# B&R Automation Studio project BenchEDM_AS6 (part 7)

#### Seq_INIT_X.st - not listed in the package file held
```iecst
ACTION Seq_INIT_X:

	TC_Seq_Add(ADR(JSONStrings),ADR('{"driver":"AB","inst":"VX_0","type":"C","ident":"ERRORRESET","enable":"TRUE"}'));
	TC_Seq_Add(ADR(JSONStrings),ADR('{"driver":"AB","inst":"VX_0","type":"W","ident":"NOERROR","time":"10.0"}'));
	TC_Seq_Add(ADR(JSONStrings),ADR('{"driver":"AB","inst":"VX_0","type":"C","ident":"ERRORRESET","enable":"FALSE"}'));
	TC_Seq_Add(ADR(JSONStrings),ADR('{"driver":"AB","inst":"VX_0","type":"M","ident":"ERROR","enable":"TRUE","sev":"4","time":"0.0"}'));
	TC_Seq_Add(ADR(JSONStrings),ADR('{"driver":"AB","inst":"VX_0","type":"W","ident":"READYTOPOWERON","time":"10.0"}'));
	TC_Seq_Add(ADR(JSONStrings),ADR('{"driver":"AB","inst":"VX_0","type":"C","ident":"POWER","enable":"TRUE"}'));
	TC_Seq_Add(ADR(JSONStrings),ADR('{"driver":"AB","inst":"VX_0","type":"W","ident":"POWERON","time":"5.0"}'));
	TC_Seq_Add(ADR(JSONStrings),ADR('{"driver":"AB","inst":"VX_0","type":"M","ident":"NOTPOWERON","enable":"TRUE","sev":"4","time":"0.0"}'));
	TC_Seq_Add(ADR(JSONStrings),ADR('{"driver":"AB","inst":"VX_0","type":"C","ident":"HOME","enable":"TRUE"}'));
	TC_Seq_Add(ADR(JSONStrings),ADR('{"driver":"AB","inst":"VX_0","type":"W","ident":"ISHOMED","time":"5.0"}'));
	TC_Seq_Add(ADR(JSONStrings),ADR('{"driver":"AB","inst":"VX_0","type":"C","ident":"HOME","enable":"FALSE"}'));

	TC_Seq_Add(ADR(JSONStrings),ADR('{"driver":"AB","inst":"RX0_0","type":"C","ident":"ERRORRESET","enable":"TRUE"}'));
	TC_Seq_Add(ADR(JSONStrings),ADR('{"driver":"AB","inst":"RX0_0","type":"W","ident":"NOERROR","time":"10.0"}'));
	TC_Seq_Add(ADR(JSONStrings),ADR('{"driver":"AB","inst":"RX0_0","type":"C","ident":"ERRORRESET","enable":"FALSE"}'));
	TC_Seq_Add(ADR(JSONStrings),ADR('{"driver":"AB","inst":"RX0_0","type":"M","ident":"ERROR","enable":"TRUE","sev":"4","time":"0.0"}'));
	TC_Seq_Add(ADR(JSONStrings),ADR('{"driver":"AB","inst":"RX0_0","type":"W","ident":"READYTOPOWERON","time":"10.0"}'));
	TC_Seq_Add(ADR(JSONStrings),ADR('{"driver":"AB","inst":"RX0_0","type":"C","ident":"POWER","enable":"TRUE"}'));
	TC_Seq_Add(ADR(JSONStrings),ADR('{"driver":"AB","inst":"RX0_0","type":"W","ident":"POWERON","time":"5.0"}'));
	TC_Seq_Add(ADR(JSONStrings),ADR('{"driver":"AB","inst":"RX0_0","type":"M","ident":"NOTPOWERON","enable":"TRUE","sev":"4","time":"0.0"}'));
	TC_Seq_Add(ADR(JSONStrings),ADR('{"driver":"AB","inst":"RX0_0","type":"C","ident":"HOME","enable":"TRUE"}'));
	TC_Seq_Add(ADR(JSONStrings),ADR('{"driver":"AB","inst":"RX0_0","type":"W","ident":"ISHOMED","time":"5.0"}'));
	TC_Seq_Add(ADR(JSONStrings),ADR('{"driver":"AB","inst":"RX0_0","type":"C","ident":"HOME","enable":"FALSE"}'));

	TC_Seq_Add(ADR(JSONStrings),ADR('{"driver":"CS","inst":"RX0_0","type":"C","ident":"ERRORRESET","enable":"TRUE"}'));
	TC_Seq_Add(ADR(JSONStrings),ADR('{"driver":"CS","inst":"RX0_0","type":"W","ident":"NOERROR","time":"10.0"}'));
	TC_Seq_Add(ADR(JSONStrings),ADR('{"driver":"CS","inst":"RX0_0","type":"C","ident":"ERRORRESET","enable":"FALSE"}'));
	TC_Seq_Add(ADR(JSONStrings),ADR('{"driver":"CS","inst":"RX0_0","type":"M","ident":"ERROR","enable":"TRUE","sev":"4","time":"0.0"}'));
	TC_Seq_Add(ADR(JSONStrings),ADR('{"driver":"CS","inst":"RX0_0","type":"W","ident":"AXISREADY","time":"10.0"}'));
	TC_Seq_Add(ADR(JSONStrings),ADR('{"driver":"CS","inst":"RX0_0","type":"C","ident":"MOVECYCLICPOSITION","enable":"TRUE","par":{"CyclicPositionSource":"<SD>0"}}'));
	TC_Seq_Add(ADR(JSONStrings),ADR('{"driver":"CS","inst":"RX0_0","type":"W","ident":"MOVECYCLICPOSITIONACTIVE","time":"10.0"}'));
	TC_Seq_Add(ADR(JSONStrings),ADR('{"driver":"CS","inst":"RX0_0","type":"M","ident":"NOTMOVECYCLICPOSITIONACTIVE","enable":"TRUE","sev":"4","time":"0.0"}'));

END_ACTION
```

#### Seq_INIT_Y.st - not listed in the package file held
```iecst
ACTION Seq_INIT_Y:

	TC_Seq_Add(ADR(JSONStrings),ADR('{"driver":"AB","inst":"VY_0","type":"C","ident":"ERRORRESET","enable":"TRUE"}'));
	TC_Seq_Add(ADR(JSONStrings),ADR('{"driver":"AB","inst":"VY_0","type":"W","ident":"NOERROR","time":"10.0"}'));
	TC_Seq_Add(ADR(JSONStrings),ADR('{"driver":"AB","inst":"VY_0","type":"C","ident":"ERRORRESET","enable":"FALSE"}'));
	TC_Seq_Add(ADR(JSONStrings),ADR('{"driver":"AB","inst":"VY_0","type":"M","ident":"ERROR","enable":"TRUE","sev":"4","time":"0.0"}'));
	TC_Seq_Add(ADR(JSONStrings),ADR('{"driver":"AB","inst":"VY_0","type":"W","ident":"READYTOPOWERON","time":"10.0"}'));
	TC_Seq_Add(ADR(JSONStrings),ADR('{"driver":"AB","inst":"VY_0","type":"C","ident":"POWER","enable":"TRUE"}'));
	TC_Seq_Add(ADR(JSONStrings),ADR('{"driver":"AB","inst":"VY_0","type":"W","ident":"POWERON","time":"5.0"}'));
	TC_Seq_Add(ADR(JSONStrings),ADR('{"driver":"AB","inst":"VY_0","type":"M","ident":"NOTPOWERON","enable":"TRUE","sev":"4","time":"0.0"}'));
	TC_Seq_Add(ADR(JSONStrings),ADR('{"driver":"AB","inst":"VY_0","type":"C","ident":"HOME","enable":"TRUE"}'));
	TC_Seq_Add(ADR(JSONStrings),ADR('{"driver":"AB","inst":"VY_0","type":"W","ident":"ISHOMED","time":"5.0"}'));
	TC_Seq_Add(ADR(JSONStrings),ADR('{"driver":"AB","inst":"VY_0","type":"C","ident":"HOME","enable":"FALSE"}'));

	TC_Seq_Add(ADR(JSONStrings),ADR('{"driver":"AB","inst":"RY0_0","type":"C","ident":"ERRORRESET","enable":"TRUE"}'));
	TC_Seq_Add(ADR(JSONStrings),ADR('{"driver":"AB","inst":"RY0_0","type":"W","ident":"NOERROR","time":"10.0"}'));
	TC_Seq_Add(ADR(JSONStrings),ADR('{"driver":"AB","inst":"RY0_0","type":"C","ident":"ERRORRESET","enable":"FALSE"}'));
	TC_Seq_Add(ADR(JSONStrings),ADR('{"driver":"AB","inst":"RY0_0","type":"M","ident":"ERROR","enable":"TRUE","sev":"4","time":"0.0"}'));
	TC_Seq_Add(ADR(JSONStrings),ADR('{"driver":"AB","inst":"RY0_0","type":"W","ident":"READYTOPOWERON","time":"10.0"}'));
	TC_Seq_Add(ADR(JSONStrings),ADR('{"driver":"AB","inst":"RY0_0","type":"C","ident":"POWER","enable":"TRUE"}'));
	TC_Seq_Add(ADR(JSONStrings),ADR('{"driver":"AB","inst":"RY0_0","type":"W","ident":"POWERON","time":"5.0"}'));
	TC_Seq_Add(ADR(JSONStrings),ADR('{"driver":"AB","inst":"RY0_0","type":"M","ident":"NOTPOWERON","enable":"TRUE","sev":"4","time":"0.0"}'));
	TC_Seq_Add(ADR(JSONStrings),ADR('{"driver":"AB","inst":"RY0_0","type":"C","ident":"HOME","enable":"TRUE"}'));
	TC_Seq_Add(ADR(JSONStrings),ADR('{"driver":"AB","inst":"RY0_0","type":"W","ident":"ISHOMED","time":"5.0"}'));
	TC_Seq_Add(ADR(JSONStrings),ADR('{"driver":"AB","inst":"RY0_0","type":"C","ident":"HOME","enable":"FALSE"}'));

	TC_Seq_Add(ADR(JSONStrings),ADR('{"driver":"CS","inst":"RY0_0","type":"C","ident":"ERRORRESET","enable":"TRUE"}'));
	TC_Seq_Add(ADR(JSONStrings),ADR('{"driver":"CS","inst":"RY0_0","type":"W","ident":"NOERROR","time":"10.0"}'));
	TC_Seq_Add(ADR(JSONStrings),ADR('{"driver":"CS","inst":"RY0_0","type":"C","ident":"ERRORRESET","enable":"FALSE"}'));
	TC_Seq_Add(ADR(JSONStrings),ADR('{"driver":"CS","inst":"RY0_0","type":"M","ident":"ERROR","enable":"TRUE","sev":"4","time":"0.0"}'));
	TC_Seq_Add(ADR(JSONStrings),ADR('{"driver":"CS","inst":"RY0_0","type":"W","ident":"AXISREADY","time":"10.0"}'));
	TC_Seq_Add(ADR(JSONStrings),ADR('{"driver":"CS","inst":"RY0_0","type":"C","ident":"MOVECYCLICPOSITION","enable":"TRUE","par":{"CyclicPositionSource":"<SD>0"}}'));
	TC_Seq_Add(ADR(JSONStrings),ADR('{"driver":"CS","inst":"RY0_0","type":"W","ident":"MOVECYCLICPOSITIONACTIVE","time":"10.0"}'));
	TC_Seq_Add(ADR(JSONStrings),ADR('{"driver":"CS","inst":"RY0_0","type":"M","ident":"NOTMOVECYCLICPOSITIONACTIVE","enable":"TRUE","sev":"4","time":"0.0"}'));

END_ACTION
```

#### Seq_INIT_Z.st - not listed in the package file held
```iecst
ACTION Seq_INIT_Z:

	TC_Seq_Add(ADR(JSONStrings),ADR('{"driver":"AB","inst":"VZ_0","type":"C","ident":"ERRORRESET","enable":"TRUE"}'));
	TC_Seq_Add(ADR(JSONStrings),ADR('{"driver":"AB","inst":"VZ_0","type":"W","ident":"NOERROR","time":"10.0"}'));
	TC_Seq_Add(ADR(JSONStrings),ADR('{"driver":"AB","inst":"VZ_0","type":"C","ident":"ERRORRESET","enable":"FALSE"}'));
	TC_Seq_Add(ADR(JSONStrings),ADR('{"driver":"AB","inst":"VZ_0","type":"M","ident":"ERROR","enable":"TRUE","sev":"4","time":"0.0"}'));
	TC_Seq_Add(ADR(JSONStrings),ADR('{"driver":"AB","inst":"VZ_0","type":"W","ident":"READYTOPOWERON","time":"10.0"}'));
	TC_Seq_Add(ADR(JSONStrings),ADR('{"driver":"AB","inst":"VZ_0","type":"C","ident":"POWER","enable":"TRUE"}'));
	TC_Seq_Add(ADR(JSONStrings),ADR('{"driver":"AB","inst":"VZ_0","type":"W","ident":"POWERON","time":"5.0"}'));
	TC_Seq_Add(ADR(JSONStrings),ADR('{"driver":"AB","inst":"VZ_0","type":"M","ident":"NOTPOWERON","enable":"TRUE","sev":"4","time":"0.0"}'));
	TC_Seq_Add(ADR(JSONStrings),ADR('{"driver":"AB","inst":"VZ_0","type":"C","ident":"HOME","enable":"TRUE"}'));
	TC_Seq_Add(ADR(JSONStrings),ADR('{"driver":"AB","inst":"VZ_0","type":"W","ident":"ISHOMED","time":"5.0"}'));
	TC_Seq_Add(ADR(JSONStrings),ADR('{"driver":"AB","inst":"VZ_0","type":"C","ident":"HOME","enable":"FALSE"}'));

	TC_Seq_Add(ADR(JSONStrings),ADR('{"driver":"AB","inst":"RZ0_0","type":"C","ident":"ERRORRESET","enable":"TRUE"}'));
	TC_Seq_Add(ADR(JSONStrings),ADR('{"driver":"AB","inst":"RZ0_0","type":"W","ident":"NOERROR","time":"10.0"}'));
	TC_Seq_Add(ADR(JSONStrings),ADR('{"driver":"AB","inst":"RZ0_0","type":"C","ident":"ERRORRESET","enable":"FALSE"}'));
	TC_Seq_Add(ADR(JSONStrings),ADR('{"driver":"AB","inst":"RZ0_0","type":"M","ident":"ERROR","enable":"TRUE","sev":"4","time":"0.0"}'));
	TC_Seq_Add(ADR(JSONStrings),ADR('{"driver":"AB","inst":"RZ0_0","type":"W","ident":"READYTOPOWERON","time":"10.0"}'));
	TC_Seq_Add(ADR(JSONStrings),ADR('{"driver":"AB","inst":"RZ0_0","type":"C","ident":"POWER","enable":"TRUE"}'));
	TC_Seq_Add(ADR(JSONStrings),ADR('{"driver":"AB","inst":"RZ0_0","type":"W","ident":"POWERON","time":"5.0"}'));
	TC_Seq_Add(ADR(JSONStrings),ADR('{"driver":"AB","inst":"RZ0_0","type":"M","ident":"NOTPOWERON","enable":"TRUE","sev":"4","time":"0.0"}'));
	TC_Seq_Add(ADR(JSONStrings),ADR('{"driver":"AB","inst":"RZ0_0","type":"C","ident":"HOME","enable":"TRUE"}'));
	TC_Seq_Add(ADR(JSONStrings),ADR('{"driver":"AB","inst":"RZ0_0","type":"W","ident":"ISHOMED","time":"5.0"}'));
	TC_Seq_Add(ADR(JSONStrings),ADR('{"driver":"AB","inst":"RZ0_0","type":"C","ident":"HOME","enable":"FALSE"}'));

	TC_Seq_Add(ADR(JSONStrings),ADR('{"driver":"CS","inst":"RZ0_0","type":"C","ident":"ERRORRESET","enable":"TRUE"}'));
	TC_Seq_Add(ADR(JSONStrings),ADR('{"driver":"CS","inst":"RZ0_0","type":"W","ident":"NOERROR","time":"10.0"}'));
	TC_Seq_Add(ADR(JSONStrings),ADR('{"driver":"CS","inst":"RZ0_0","type":"C","ident":"ERRORRESET","enable":"FALSE"}'));
	TC_Seq_Add(ADR(JSONStrings),ADR('{"driver":"CS","inst":"RZ0_0","type":"M","ident":"ERROR","enable":"TRUE","sev":"4","time":"0.0"}'));
	TC_Seq_Add(ADR(JSONStrings),ADR('{"driver":"CS","inst":"RZ0_0","type":"W","ident":"AXISREADY","time":"10.0"}'));
	TC_Seq_Add(ADR(JSONStrings),ADR('{"driver":"CS","inst":"RZ0_0","type":"C","ident":"MOVECYCLICPOSITION","enable":"TRUE","par":{"CyclicPositionSource":"<SD>0"}}'));
	TC_Seq_Add(ADR(JSONStrings),ADR('{"driver":"CS","inst":"RZ0_0","type":"W","ident":"MOVECYCLICPOSITIONACTIVE","time":"10.0"}'));
	TC_Seq_Add(ADR(JSONStrings),ADR('{"driver":"CS","inst":"RZ0_0","type":"M","ident":"NOTMOVECYCLICPOSITIONACTIVE","enable":"TRUE","sev":"4","time":"0.0"}'));

END_ACTION
```

### Program Logical/Process/OutputMan (IEC)

#### Main.st - Init, cyclic, exit code
```iecst
PROGRAM _INIT

END_PROGRAM

PROGRAM _CYCLIC

	OMD_CN;
	OMD_AB;
	OMD_CS;
	OMD_MR;
	OMD_BX;
	gDriver.ResetAll := FALSE;

//BX18

	IF (gIO.BX18.TC_IO_DO_Enable.Forcing.On AND gIO.BX18.TC_IO_DO_Enable.Forcing.Off) OR NOT gIO.ForceEnable THEN
		gIO.BX18.TC_IO_DO_Enable.Forcing.On									:= FALSE;
		gIO.BX18.TC_IO_DO_Enable.Forcing.Off								:= FALSE;
	END_IF;
	gIO.BX18.TC_IO_DO_Enable(Par := gPar.IO.BX18.TC_IO_DO_Enable);

	IF (gIO.BX18.TC_IO_DO_ISOFreqMode.Forcing.On AND gIO.BX18.TC_IO_DO_ISOFreqMode.Forcing.Off) OR NOT gIO.ForceEnable THEN
		gIO.BX18.TC_IO_DO_ISOFreqMode.Forcing.On							:= FALSE;
		gIO.BX18.TC_IO_DO_ISOFreqMode.Forcing.Off							:= FALSE;
	END_IF;
	gIO.BX18.TC_IO_DO_ISOFreqMode(Par := gPar.IO.BX18.TC_IO_DO_ISOFreqMode);

	IF (gIO.BX18.TC_IO_DO_EdgeFindMode.Forcing.On AND gIO.BX18.TC_IO_DO_EdgeFindMode.Forcing.Off) OR NOT gIO.ForceEnable THEN
		gIO.BX18.TC_IO_DO_EdgeFindMode.Forcing.On							:= FALSE;
		gIO.BX18.TC_IO_DO_EdgeFindMode.Forcing.Off							:= FALSE;
	END_IF;
	gIO.BX18.TC_IO_DO_EdgeFindMode(Par := gPar.IO.BX18.TC_IO_DO_EdgeFindMode);

	IF (gIO.BX18.TC_IO_DO_ElectrodePositiveMode.Forcing.On AND gIO.BX18.TC_IO_DO_ElectrodePositiveMode.Forcing.Off) OR NOT gIO.ForceEnable THEN
		gIO.BX18.TC_IO_DO_ElectrodePositiveMode.Forcing.On					:= FALSE;
		gIO.BX18.TC_IO_DO_ElectrodePositiveMode.Forcing.Off					:= FALSE;
	END_IF;
	gIO.BX18.TC_IO_DO_ElectrodePositiveMode(Par := gPar.IO.BX18.TC_IO_DO_ElectrodePositiveMode);

	IF (gIO.BX18.TC_IO_DO_ChangeRequest.Forcing.On AND gIO.BX18.TC_IO_DO_ChangeRequest.Forcing.Off) OR NOT gIO.ForceEnable THEN
		gIO.BX18.TC_IO_DO_ChangeRequest.Forcing.On							:= FALSE;
		gIO.BX18.TC_IO_DO_ChangeRequest.Forcing.Off							:= FALSE;
	END_IF;
	gIO.BX18.TC_IO_DO_ChangeRequest(Par := gPar.IO.BX18.TC_IO_DO_ChangeRequest);

	IF (gIO.BX18.TC_IO_AO_OnTime.Forcing.On AND gIO.BX18.TC_IO_AO_OnTime.Forcing.Off) OR NOT gIO.ForceEnable THEN
		gIO.BX18.TC_IO_AO_OnTime.Forcing.On									:= FALSE;
		gIO.BX18.TC_IO_AO_OnTime.Forcing.Off								:= FALSE;
	END_IF;
	gIO.BX18.TC_IO_AO_OnTime(Par := gPar.IO.BX18.TC_IO_AO_OnTime, VarType := TC_IO_ANALOG_TYPE_UINT);

	IF (gIO.BX18.TC_IO_AO_OffTime.Forcing.On AND gIO.BX18.TC_IO_AO_OffTime.Forcing.Off) OR NOT gIO.ForceEnable THEN
		gIO.BX18.TC_IO_AO_OffTime.Forcing.On								:= FALSE;
		gIO.BX18.TC_IO_AO_OffTime.Forcing.Off								:= FALSE;
	END_IF;
	gIO.BX18.TC_IO_AO_OffTime(Par := gPar.IO.BX18.TC_IO_AO_OffTime, VarType := TC_IO_ANALOG_TYPE_UINT);

	IF (gIO.BX18.TC_IO_AO_Current.Forcing.On AND gIO.BX18.TC_IO_AO_Current.Forcing.Off) OR NOT gIO.ForceEnable THEN
		gIO.BX18.TC_IO_AO_Current.Forcing.On								:= FALSE;
		gIO.BX18.TC_IO_AO_Current.Forcing.Off								:= FALSE;
	END_IF;
	gIO.BX18.TC_IO_AO_Current(Par := gPar.IO.BX18.TC_IO_AO_Current, VarType := TC_IO_ANALOG_TYPE_UINT);

	gIO.BX18.Outputs_control.0												:= gIO.BX18.TC_IO_DO_Enable.Signal.IOMapping;
	gIO.BX18.Outputs_control.1												:= gIO.BX18.TC_IO_DO_ISOFreqMode.Signal.IOMapping;
	gIO.BX18.Outputs_control.2												:= gIO.BX18.TC_IO_DO_EdgeFindMode.Signal.IOMapping;
	gIO.BX18.Outputs_control.3												:= gIO.BX18.TC_IO_DO_ElectrodePositiveMode.Signal.IOMapping;
	gIO.BX18.Outputs_control.4												:= gIO.BX18.TC_IO_DO_ChangeRequest.Signal.IOMapping;
	gIO.BX18.Outputs_onTime													:= gIO.BX18.TC_IO_AO_OnTime.Signal.IOMapping.VarUINT;
	gIO.BX18.Outputs_offTime												:= gIO.BX18.TC_IO_AO_OffTime.Signal.IOMapping.VarUINT;
	gIO.BX18.Outputs_current												:= gIO.BX18.TC_IO_AO_Current.Signal.IOMapping.VarUINT;
//Motion
	gIO.Motion.SetPosition 													:= LREAL_TO_DINT(gDriver.AB[DRIVER_INST_AB_RZ_0_0].Status.Position*200.0); //200.0 is the scaling to get 1mm travel for 1000 dip switch setting on stepper drive
	gIO.Motion.StepDelay 													:= STEPDELAY;
	gIO.Motion.ENABLE														:= gIO.Motion.ModuleOK;
	gIO.Motion.SwitchedOn													:= gIO.Motion.ENABLED AND gIO.Motion.SwitchOn AND gIO.Safety.TC_IO_DI_ESTOP.Signal.Filtered;
	gIO.Motion.Home															:= EDGEPOS(gDriver.AB[DRIVER_INST_AB_RZ_0_0].MpAxisBasic_0.IsHomed);
//MbRTU VFDs
	FOR i := 0 TO MAX_VFD_IDX DO
		gIO.VFD[i].DataWrite[0] := gIO.VFD[i].CMD;
		gIO.VFD[i].DataWrite[1] := gIO.VFD[i].LFRD;
		FOR j := 0 TO MAX_VFD_DATA_READ_IDX DO
			gIO.VFD[i].EventRead[j]											:= TRUE;
		END_FOR;
		gIO.VFD[i].CTON_AutoWrite(IN := NOT gIO.VFD[i].CTON_AutoWrite.Q, PT := T#500ms);
		FOR j := 0 TO MAX_VFD_DATA_WRITE_IDX DO
			IF gIO.VFD[i].DataWriteCmp[j] <> gIO.VFD[i].DataWrite[j] OR gIO.VFD[i].CTON_AutoWrite.Q THEN
				gIO.VFD[i].EventWrite[j]									:= TRUE;
				gIO.VFD[i].DataWriteCmp[j] 									:= gIO.VFD[i].DataWrite[j];
			END_IF;
		END_FOR;
		gIO.VFD[i].ETA := gIO.VFD[i].DataRead[0];
		gIO.VFD[i].RFRD := gIO.VFD[i].DataRead[1];
		gIO.VFD[i].LFT := gIO.VFD[i].DataRead[2];
	END_FOR;

END_PROGRAM

PROGRAM _EXIT

END_PROGRAM
```

#### OMD_IN.st
```iecst
ACTION OMD_IN:

//	FOR i := 0 TO MAX_DRIVER_IN_IDX DO
//		IF NOT gDriver.IN[i].FirstScanComplete THEN
//			gDriver.IN[i].FirstScanComplete 													:= TRUE;
//
//			gDriver.IN[i].DefaultPar.DI_Estop_Par.FilterOnTime									:= 50.0;							//LR
//			gDriver.IN[i].DefaultPar.DI_Estop_Par.FilterOffTime									:= 50.0;							//LR
//			gDriver.IN[i].DefaultPar.DI_Estop_Par.InvertedIOMapping								:= FALSE;							//BO
//			gDriver.IN[i].DefaultPar.DI_Estop_Forcing.On										:= FALSE;							//BO
//			gDriver.IN[i].DefaultPar.DI_Estop_Forcing.Off										:= FALSE;							//BO
//			gDriver.IN[i].DefaultPar.DI_Estop_Sim.Active										:= gSim.Full OR gSim.IO;			//BO
//			gDriver.IN[i].DefaultPar.DI_Estop_Sim.Logical										:= FALSE;							//BO
//
//			brsmemcpy(ADR(gDriver.IN[i].Par),ADR(gDriver.IN[i].DefaultPar),SIZEOF(gDriver.IN[i].Par));
//		END_IF;
//
//		brsmemset(ADR(gDriver.IN[i].Sev),0,SIZEOF(gDriver.IN[i].Sev));
//		brsmemset(ADR(gDriver.IN[i].Status),0,SIZEOF(gDriver.IN[i].Status));
//		FOR j := 0 TO MAX_DRIVER_IN_MON_IDX DO
//			IF gDriver.IN[i].Par.Mon[j].Enable THEN
//				IF gDriver.IN[i].Mon[j] THEN
//					gDriver.IN[i].CTON_Mon[j](IN := TRUE, PT := LREAL_TO_TIME(gDriver.IN[i].Par.Mon[j].Time*1000.0));
//					IF gDriver.IN[i].CTON_Mon[j].Q THEN
//						gDriver.IN[i].Sev[j] := gDriver.IN[i].Par.Mon[j].Sev;
//						IF gDriver.IN[i].Status.Severity < gDriver.IN[i].Sev[j] THEN
//							gDriver.IN[i].Status.Severity := gDriver.IN[i].Sev[j];
//						END_IF;
//					END_IF;
//				ELSE
//					gDriver.IN[i].CTON_Mon[j](IN := FALSE);
//					gDriver.IN[i].Sev[j] := 0;
//				END_IF;
//			ELSE
//				gDriver.IN[i].CTON_Mon[j](IN := FALSE);
//				gDriver.IN[i].Sev[j] := 0;
//			END_IF;
//		END_FOR;
//		IF gDriver.IN[i].Cmd[C_IN_RESET] THEN
//			gDriver.IN[i].Cmd[C_IN_RESET] := FALSE;
//			brsmemset(ADR(gDriver.IN[i].Cmd),0,SIZEOF(gDriver.IN[i].Cmd));
//			brsmemset(ADR(gDriver.IN[i].Sev),0,SIZEOF(gDriver.IN[i].Sev));
//			brsmemset(ADR(gDriver.IN[i].Status),0,SIZEOF(gDriver.IN[i].Status));
//			brsmemcpy(ADR(gDriver.IN[i].Par),ADR(gDriver.IN[i].DefaultPar),SIZEOF(gDriver.IN[i].Par));
//		END_IF;
//		IF gDriver.IN[i].Cmd[C_IN_CLEARCMD] THEN
//			gDriver.IN[i].Cmd[C_IN_CLEARCMD] := FALSE;
//			brsmemset(ADR(gDriver.IN[i].Cmd),0,SIZEOF(gDriver.IN[i].Cmd));
//		END_IF;
//		IF gDriver.IN[i].Cmd[C_IN_CLEARMON] THEN
//			gDriver.IN[i].Cmd[C_IN_CLEARMON] := FALSE;
//			brsmemset(ADR(gDriver.IN[i].Status.Severity),0,SIZEOF(gDriver.IN[i].Status.Severity));
//			brsmemset(ADR(gDriver.IN[i].Sev),0,SIZEOF(gDriver.IN[i].Sev));
//			brsmemset(ADR(gDriver.IN[i].Par.Mon),0,SIZEOF(gDriver.IN[i].Par.Mon));
//		END_IF;
//		IF gDriver.IN[i].Cmd[C_IN_DEFAULTMON] THEN
//			gDriver.IN[i].Cmd[C_IN_DEFAULTMON] := FALSE;
//			brsmemcpy(ADR(gDriver.IN[i].Par.Mon),ADR(gDriver.IN[i].DefaultPar.Mon),SIZEOF(gDriver.IN[i].Par.Mon));
//		END_IF;
//		IF gDriver.IN[i].Cmd[C_IN_CLEARPAR] THEN
//			gDriver.IN[i].Cmd[C_IN_CLEARPAR] := FALSE;
//			brsmemset(ADR(gDriver.IN[i].Par),0,SIZEOF(gDriver.IN[i].Par));
//		END_IF;
//		IF gDriver.IN[i].Cmd[C_IN_DEFAULTPAR] THEN
//			gDriver.IN[i].Cmd[C_IN_DEFAULTPAR] := FALSE;
//			brsmemcpy(ADR(gDriver.IN[i].Par),ADR(gDriver.IN[i].DefaultPar),SIZEOF(gDriver.IN[i].Par));
//		END_IF;
//		IF gDriver.IN[i].Cmd[C_IN_FORCEENABLE] THEN
//			gDriver.IN[i].Cmd[C_IN_FORCEENABLE] := FALSE;
//			gDriver.IN[i].Par.ForceEnable := TRUE;
//		END_IF;
//		IF gDriver.IN[i].Cmd[C_IN_FORCEDISABLE] THEN
//			gDriver.IN[i].Cmd[C_IN_FORCEDISABLE] := FALSE;
//			gDriver.IN[i].Par.ForceEnable := FALSE;
//		END_IF;
//
//		IF NOT gDriver.IN[i].Par.ForceEnable OR (gDriver.IN[i].Par.DI_Estop_Forcing.On AND gDriver.IN[i].Par.DI_Estop_Forcing.Off) THEN
//			gDriver.IN[i].Par.DI_Estop_Forcing.On := FALSE;
//			gDriver.IN[i].Par.DI_Estop_Forcing.Off := FALSE;
//		END_IF;
//		gDriver.IN[i].DI_Estop(Forcing := gDriver.IN[i].Par.DI_Estop_Forcing, Par := gDriver.IN[i].Par.DI_Estop_Par, Sim := gDriver.IN[i].Par.DI_Estop_Sim);
//
//		gDriver.IN[i].Wait[W_IN_DI_ESTOP]				:= BOOL_TO_DINT(NOT gDriver.IN[i].DI_Estop.Signal.Filtered);
//
//		gDriver.IN[i].Mon[M_IN_ERROR]					:= gDriver.IN[i].MpAxisBasic_0.Error;
//	END_FOR;
//
////	McSwitchEnum :
////	(
////		mcSWITCH_OFF := 0,		 						(*State/Behavior selection switched off*)
////		mcSWITCH_ON := 1			 					(*State/Behavior selection switched on*)
////	);

END_ACTION
```

#### OMD_CN.st
```iecst
ACTION OMD_CN:

	gDriver.CN[DRIVER_INST_CN_0].MpLinkADR 																:= ADR(gCNC);
	gDriver.CN[DRIVER_INST_CN_0].OverrideSetpoint[0]													:= 100.0;
	gDriver.CN[DRIVER_INST_CN_0].OverrideSetpoint[1]													:= gDriver.BX[DRIVER_INST_BX_0].Status.OverrideFactor;
	gDriver.CN[DRIVER_INST_CN_0].RapidOverrideSetpoint[0]												:= 100.0;
	gDriver.CN[DRIVER_INST_CN_0].FeedrateOverrideSetpoint[0]											:= 100.0;

	FOR i := 0 TO MAX_DRIVER_CN_IDX DO
		IF NOT gDriver.CN[i].FirstScanComplete THEN
			gDriver.CN[i].FirstScanComplete 															:= TRUE;

			gDriver.CN[i].DefaultPar.CN.Block															:= '';								//ST
			gDriver.CN[i].DefaultPar.CN.Jog.CoordSystem													:= 0;								//UD
			gDriver.CN[i].DefaultPar.CN.Jog.PathLimits.Acceleration										:= 50.0;							//RR
			gDriver.CN[i].DefaultPar.CN.Jog.PathLimits.Deceleration										:= 50.0;							//RR
			gDriver.CN[i].DefaultPar.CN.Jog.PathLimits.Jerk												:= 0.0;								//RR
			gDriver.CN[i].DefaultPar.CN.Jog.PathLimits.Velocity											:= 10.0;							//RR
			gDriver.CN[i].DefaultPar.CN.MoveProgramOptions.InitProgram									:= '';								//ST
			gDriver.CN[i].DefaultPar.CN.MoveProgramOptions.RepositioningParameter.AxisVelocityFactor	:= 10.0;							//RR
			gDriver.CN[i].DefaultPar.CN.MoveProgramOptions.RepositioningParameter.String				:= '';								//ST
			gDriver.CN[i].DefaultPar.CN.MoveProgramOptions.RepositioningParameter.Type					:= mcPRGRP_SINGLE_AXIS;				//McPrgAxesReposTypeEnum
			gDriver.CN[i].DefaultPar.CN.MoveProgramOptions.SaveRestartData								:= mcSWITCH_OFF;					//McSwitchEnum
			gDriver.CN[i].DefaultPar.CN.MoveProgramOptions.StartMode									:= mcPRGSM_NON_MODAL;				//McPrgStartModeEnum
			gDriver.CN[i].DefaultPar.CN.MoveProgramOptions.StartPointParameter							:= 0.0;								//LR
			gDriver.CN[i].DefaultPar.CN.MoveProgramOptions.StartPointType								:= mcPRGSP_STANDARD;				//McPrgStartPointEnum
			gDriver.CN[i].DefaultPar.CN.ProgramName														:= '';								//ST
			gDriver.CN[i].DefaultPar.FeedrateOverrideSource												:= 0;								//SD
			gDriver.CN[i].DefaultPar.OverrideSource														:= 0;								//SD
			gDriver.CN[i].DefaultPar.RapidOverrideSource												:= 0;								//SD
			brsmemcpy(ADR(gDriver.CN[i].Par),ADR(gDriver.CN[i].DefaultPar),SIZEOF(gDriver.CN[i].Par));
		ELSIF NOT gDriver.CN[i].ParametersLoaded AND gMain.Services.Recipes.Out.ParametersReady THEN
			gDriver.CN[i].ParametersLoaded := TRUE;
			brsmemcpy(ADR(gDriver.CN[i].Par),ADR(gPar.Driver.CN[i]),SIZEOF(gDriver.CN[i].Par));
		END_IF;

		brsmemset(ADR(gDriver.CN[i].Sev),0,SIZEOF(gDriver.CN[i].Sev));
		brsmemset(ADR(gDriver.CN[i].Status),0,SIZEOF(gDriver.CN[i].Status));
		FOR j := 0 TO MAX_DRIVER_CN_MON_IDX DO
			IF gDriver.CN[i].Par.Mon[j].Enable THEN
				IF gDriver.CN[i].Mon[j] THEN
					gDriver.CN[i].CTON_Mon[j](IN := TRUE, PT := LREAL_TO_TIME(gDriver.CN[i].Par.Mon[j].Time*1000.0));
					IF gDriver.CN[i].CTON_Mon[j].Q THEN
						gDriver.CN[i].Sev[j] := gDriver.CN[i].Par.Mon[j].Sev;
						IF gDriver.CN[i].Status.Severity < gDriver.CN[i].Sev[j] THEN
							gDriver.CN[i].Status.Severity := gDriver.CN[i].Sev[j];
						END_IF;
					END_IF;
				ELSE
					gDriver.CN[i].CTON_Mon[j](IN := FALSE);
					gDriver.CN[i].Sev[j] := 0;
				END_IF;
			ELSE
				gDriver.CN[i].CTON_Mon[j](IN := FALSE);
				gDriver.CN[i].Sev[j] := 0;
			END_IF;
		END_FOR;
		IF gDriver.CN[i].Cmd[C_CN_RESET] OR gDriver.ResetAll THEN
			gDriver.CN[i].Cmd[C_CN_RESET] := FALSE;
			brsmemset(ADR(gDriver.CN[i].Mon),0,SIZEOF(gDriver.CN[i].Mon));
			brsmemset(ADR(gDriver.CN[i].Cmd),0,SIZEOF(gDriver.CN[i].Cmd));
			brsmemset(ADR(gDriver.CN[i].Sev),0,SIZEOF(gDriver.CN[i].Sev));
			brsmemset(ADR(gDriver.CN[i].Status),0,SIZEOF(gDriver.CN[i].Status));
		END_IF;
		IF gDriver.CN[i].Cmd[C_CN_CLEARCMD] THEN
			gDriver.CN[i].Cmd[C_CN_CLEARCMD] := FALSE;
			brsmemset(ADR(gDriver.CN[i].Cmd),0,SIZEOF(gDriver.CN[i].Cmd));
		END_IF;
		IF gDriver.CN[i].Cmd[C_CN_CLEARMON] THEN
			gDriver.CN[i].Cmd[C_CN_CLEARMON] := FALSE;
			brsmemset(ADR(gDriver.CN[i].Status.Severity),0,SIZEOF(gDriver.CN[i].Status.Severity));
			brsmemset(ADR(gDriver.CN[i].Sev),0,SIZEOF(gDriver.CN[i].Sev));
			brsmemset(ADR(gDriver.CN[i].Par.Mon),0,SIZEOF(gDriver.CN[i].Par.Mon));
		END_IF;
		IF gDriver.CN[i].Cmd[C_CN_DEFAULTMON] THEN
			gDriver.CN[i].Cmd[C_CN_DEFAULTMON] := FALSE;
			brsmemcpy(ADR(gDriver.CN[i].Par.Mon),ADR(gDriver.CN[i].DefaultPar.Mon),SIZEOF(gDriver.CN[i].Par.Mon));
		END_IF;
		IF gDriver.CN[i].Cmd[C_CN_CLEARPAR] THEN
			gDriver.CN[i].Cmd[C_CN_CLEARPAR] := FALSE;
			brsmemset(ADR(gDriver.CN[i].Par),0,SIZEOF(gDriver.CN[i].Par));
		END_IF;
		IF gDriver.CN[i].Cmd[C_CN_DEFAULTPAR] THEN
			gDriver.CN[i].Cmd[C_CN_DEFAULTPAR] := FALSE;
			brsmemcpy(ADR(gDriver.CN[i].Par),ADR(gDriver.CN[i].DefaultPar),SIZEOF(gDriver.CN[i].Par));
		END_IF;
		IF gDriver.CN[i].Cmd[C_CN_SAVEPAR] THEN
			gDriver.CN[i].Cmd[C_CN_SAVEPAR] := FALSE;
			brsmemcpy(ADR(gPar.Driver.CN[i]),ADR(gDriver.CN[i].Par),SIZEOF(gDriver.CN[i].Par));
		END_IF;
		IF gDriver.CN[i].Cmd[C_CN_LOADPAR] THEN
			gDriver.CN[i].Cmd[C_CN_LOADPAR] := FALSE;
			brsmemcpy(ADR(gDriver.CN[i].Par),ADR(gPar.Driver.CN[i]),SIZEOF(gDriver.CN[i].Par));
		END_IF;

		gDriver.CN[i].MpCncFlex_0.ErrorReset							:= gDriver.CN[i].Cmd[C_CN_ERRORRESET] OR gMain.ErrorReset;
		gDriver.CN[i].MpCncFlex_0.Continue								:= gDriver.CN[i].Cmd[C_CN_CONTINUE];
		gDriver.CN[i].MpCncFlex_0.Home									:= gDriver.CN[i].Cmd[C_CN_HOME];
		gDriver.CN[i].MpCncFlex_0.Interrupt								:= gDriver.CN[i].Cmd[C_CN_INTERRUPT];
		gDriver.CN[i].MpCncFlex_0.Jog									:= gDriver.CN[i].Cmd[C_CN_JOG];
		gDriver.CN[i].MpCncFlex_0.MoveBlock								:= gDriver.CN[i].Cmd[C_CN_MOVEBLOCK];
		gDriver.CN[i].MpCncFlex_0.MoveProgram							:= gDriver.CN[i].Cmd[C_CN_MOVEPROGRAM];
		gDriver.CN[i].MpCncFlex_0.Power									:= gDriver.CN[i].Cmd[C_CN_POWER];
		gDriver.CN[i].MpCncFlex_0.SingleStep							:= gDriver.CN[i].Cmd[C_CN_SINGLESTEP];
		gDriver.CN[i].MpCncFlex_0.Stop									:= gDriver.CN[i].Cmd[C_CN_STOP];
		gDriver.CN[i].MpCncFlex_0.Update								:= gDriver.CN[i].Cmd[C_CN_UPDATE];

		gDriver.CN[i].MpCncFlex_0.Override								:= 0.0;
		IF gDriver.CN[i].Par.OverrideSource <= MAX_DRIVER_CN_SOURCE_IDX THEN
			gDriver.CN[i].MpCncFlex_0.Override							:= gDriver.CN[i].OverrideSetpoint[gDriver.CN[i].Par.OverrideSource];
		END_IF;
		gDriver.CN[i].MpCncFlex_0.RapidOverride							:= 0.0;
		IF gDriver.CN[i].Par.RapidOverrideSource <= MAX_DRIVER_CN_SOURCE_IDX THEN
			gDriver.CN[i].MpCncFlex_0.RapidOverride						:= gDriver.CN[i].RapidOverrideSetpoint[gDriver.CN[i].Par.RapidOverrideSource];
		END_IF;
		gDriver.CN[i].MpCncFlex_0.FeedrateOverride						:= 0.0;
		IF gDriver.CN[i].Par.FeedrateOverrideSource <= MAX_DRIVER_CN_SOURCE_IDX THEN
			gDriver.CN[i].MpCncFlex_0.FeedrateOverride					:= gDriver.CN[i].FeedrateOverrideSetpoint[gDriver.CN[i].Par.FeedrateOverrideSource];
		END_IF;

		gDriver.CN[i].MpCncFlex_0(MpLink := gDriver.CN[i].MpLinkADR, Enable := TRUE, Parameters := ADR(gDriver.CN[i].Par.CN));
		gDriver.CN[i].MC_GroupReadActualPosition_15_0(AxesGroup := gDriver.CN[i].MpLinkADR, Enable := TRUE, CoordSystem := mcJACS);

		gDriver.CN[i].Status.Position_mcJACS := gDriver.CN[i].MC_GroupReadActualPosition_15_0.Position;

		gDriver.CN[i].Wait[W_CN_NOERROR]								:= BOOL_TO_DINT(NOT gDriver.CN[i].MpCncFlex_0.Error);
		gDriver.CN[i].Wait[W_CN_COMMANDABORTED]							:= BOOL_TO_DINT(gDriver.CN[i].MpCncFlex_0.CommandAborted);
		gDriver.CN[i].Wait[W_CN_COMMANDBUSY]							:= BOOL_TO_DINT(gDriver.CN[i].MpCncFlex_0.CommandBusy);
		gDriver.CN[i].Wait[W_CN_UPDATEDONE]								:= BOOL_TO_DINT(gDriver.CN[i].MpCncFlex_0.UpdateDone);
		gDriver.CN[i].Wait[W_CN_INMOTION]								:= BOOL_TO_DINT(gDriver.CN[i].MpCncFlex_0.InMotion);
		gDriver.CN[i].Wait[W_CN_ISHOMED]								:= BOOL_TO_DINT(gDriver.CN[i].MpCncFlex_0.IsHomed);
		gDriver.CN[i].Wait[W_CN_MOVEACTIVE]								:= BOOL_TO_DINT(gDriver.CN[i].MpCncFlex_0.MoveActive);
		gDriver.CN[i].Wait[W_CN_MOVEDONE]								:= BOOL_TO_DINT(gDriver.CN[i].MpCncFlex_0.MoveDone);
		gDriver.CN[i].Wait[W_CN_MOVEINTERRUPTED]						:= BOOL_TO_DINT(gDriver.CN[i].MpCncFlex_0.MoveInterrupted);
		gDriver.CN[i].Wait[W_CN_POWERON]								:= BOOL_TO_DINT(gDriver.CN[i].MpCncFlex_0.PowerOn);
		gDriver.CN[i].Wait[W_CN_SINGLESTEPACTIVE]						:= BOOL_TO_DINT(gDriver.CN[i].MpCncFlex_0.SingleStepActive);
		gDriver.CN[i].Wait[W_CN_STOPPED]								:= BOOL_TO_DINT(gDriver.CN[i].MpCncFlex_0.Stopped);
		gDriver.CN[i].Wait[W_CN_COMMUNICATIONREADY]						:= BOOL_TO_DINT(gDriver.CN[i].MpCncFlex_0.Info.CommunicationReady);
		gDriver.CN[i].Wait[W_CN_READYTOPOWERON]							:= BOOL_TO_DINT(gDriver.CN[i].MpCncFlex_0.Info.ReadyToPowerOn);
		gDriver.CN[i].Wait[W_CN_WAITFORCONTINUE]						:= BOOL_TO_DINT(gDriver.CN[i].MpCncFlex_0.Info.WaitForContinue);

		gDriver.CN[i].Mon[M_CN_ERROR]									:= gDriver.CN[i].MpCncFlex_0.Error;
		gDriver.CN[i].Mon[M_CN_NOTPOWERON]								:= NOT gDriver.CN[i].MpCncFlex_0.PowerOn;
		gDriver.CN[i].Mon[M_CN_NOTMOVEACTIVE]							:= NOT gDriver.CN[i].MpCncFlex_0.MoveActive;
	END_FOR;

//	McPrgAxesReposTypeEnum :
//	(
//		mcPRGRP_SINGLE_AXIS, (*The axes are positioned by single-axis movements*)
//		mcPRGRP_PROGRAM, (*The axes are positioned by a program*)
//		mcPRGRP_SINGLE_AXIS_AUTOMATIC (*The axes are positioned automatically*)
//	);
//	McSwitchEnum :
//	(
//		mcSWITCH_OFF,					(*State/Behavior selection switched off*)
//		mcSWITCH_ON			 			(*State/Behavior selection switched on*)
//	);
//	McPrgStartModeEnum :
//	(
//		mcPRGSM_NON_MODAL, (*Non-modal start mode*)
//		mcPRGSM_MODAL, (*Modal start mode*)
//		mcPRGSM_RESTART, (*Starts the program using the saved restart data*)
//		mcPRGSM_SIMULATION, (*High-precision simulation*)
//		mcPRGSM_SIMULATION_GEOMETRY (*Geometric simulation*)
//	);
//	McPrgStartPointEnum :
//	(
//		mcPRGSP_STANDARD, (*Start at beginning*)
//		mcPRGSP_BLOCK_NUMBER, (*Start at specified block number*)
//		mcPRGSP_ABORT_LINE, (*Start at the line number at which the program aborted*)
//		mcPRGSP_ABORT_POINT, (*Start at the point where the program aborted*)
//		mcPRGSP_LINE_NUMBER := 5, (*Start at the specified line number*)
//		mcPRGSP_PATH_DISTANCE_LINE (*Start at line in which the specified path is reached*)
//	);

END_ACTION
```

#### OMD_TR.st
```iecst
ACTION OMD_TR:

//	FOR i := 0 TO MAX_DRIVER_TR_IDX DO
//		IF gIO.SpacePilot.TC_IO_DI_Button[BUTTON_ESC].Signal.EdgePosFiltered THEN
//			gDriver.TR[i].Cmd[C_TR_RESET] := TRUE;
//		END_IF;
//
//		IF gIO.SpacePilot.TC_IO_DI_Button[BUTTON_CTRL].Signal.EdgePosFiltered THEN
//			gDriver.TR[i].Cmd[C_TR_ENABLE] := NOT gDriver.TR[i].Cmd[C_TR_ENABLE];
//		END_IF;
//
//		IF gIO.SpacePilot.TC_IO_DI_Button[BUTTON_ROT].Signal.EdgePosFiltered THEN
//			gDriver.TR[i].Par.ControlMode := TR_CONTROL_MODE_ROTATE;
//		ELSIF gIO.SpacePilot.TC_IO_DI_Button[BUTTON_TRANS].Signal.EdgePosFiltered THEN
//			gDriver.TR[i].Par.ControlMode := TR_CONTROL_MODE_TRANS;
//		ELSIF gIO.SpacePilot.TC_IO_DI_Button[BUTTON_COORD].Signal.EdgePosFiltered THEN
//			gDriver.TR[i].Par.ControlMode := TR_CONTROL_MODE_COORD;
//		END_IF;
//
//		IF gIO.SpacePilot.TC_IO_DI_Button[BUTTON_PLUS].Signal.EdgePosFiltered THEN
//			gDriver.TR[i].Par.VelocityFactor := gDriver.TR[i].Par.VelocityFactor + 0.00001;
//		ELSIF gIO.SpacePilot.TC_IO_DI_Button[BUTTON_MINUS].Signal.EdgePosFiltered THEN
//			gDriver.TR[i].Par.VelocityFactor := gDriver.TR[i].Par.VelocityFactor - 0.00001;
//		END_IF;
//
//		FOR j := 0 TO MAX_AXIS_V_IDX DO
//			gDriver.TR[i].Status.InputCmd[j] := gIO.SpacePilot.TC_IO_AI_Joystick[j].Signal.Filtered;
//		END_FOR;
//
//		IF NOT gDriver.TR[i].FirstScanComplete THEN
//			gDriver.TR[i].FirstScanComplete 													:= TRUE;
//			gDriver.TR[i].DefaultPar.ControlMode												:= TR_CONTROL_MODE_COORD; 	//TR_CONTROL_MODE_ENUM
//			gDriver.TR[i].DefaultPar.Filter														:= 0.99;						//LR
//			gDriver.TR[i].DefaultPar.VelocityFactor												:= 0.00005;					//LR
//			gDriver.TR[i].DefaultPar.Gain														:= 10.0;						//RR
//			gDriver.TR[i].DefaultPar.IntegralTime												:= 0.1;						//RR
//			brsmemcpy(ADR(gDriver.TR[i].Par),ADR(gDriver.TR[i].DefaultPar),SIZEOF(gDriver.TR[i].Par));
//
//			brsmemcpy(ADR(gDriver.TR[i].Par),ADR(gDriver.TR[i].DefaultPar),SIZEOF(gDriver.TR[i].Par));
//		ELSIF NOT gDriver.TR[i].ParametersLoaded AND gMain.Services.Recipes.Out.ParametersReady THEN
//			gDriver.TR[i].ParametersLoaded := TRUE;
//			brsmemcpy(ADR(gDriver.TR[i].Par),ADR(gPar.Driver.TR[i]),SIZEOF(gDriver.TR[i].Par));
//		END_IF;
//
//		brsmemset(ADR(gDriver.TR[i].Sev),0,SIZEOF(gDriver.TR[i].Sev));
//		FOR j := 0 TO MAX_DRIVER_TR_MON_IDX DO
//			IF gDriver.TR[i].Par.Mon[j].Enable THEN
//				IF gDriver.TR[i].Mon[j] THEN
//					gDriver.TR[i].CTON_Mon[j](IN := TRUE, PT := LREAL_TO_TIME(gDriver.TR[i].Par.Mon[j].Time*1000.0));
//					IF gDriver.TR[i].CTON_Mon[j].Q THEN
//						gDriver.TR[i].Sev[j] := gDriver.TR[i].Par.Mon[j].Sev;
//						IF gDriver.TR[i].Status.Severity < gDriver.TR[i].Sev[j] THEN
//							gDriver.TR[i].Status.Severity := gDriver.TR[i].Sev[j];
//						END_IF;
//					END_IF;
//				ELSE
//					gDriver.TR[i].CTON_Mon[j](IN := FALSE);
//					gDriver.TR[i].Sev[j] := 0;
//				END_IF;
//			ELSE
//				gDriver.TR[i].CTON_Mon[j](IN := FALSE);
//				gDriver.TR[i].Sev[j] := 0;
//			END_IF;
//		END_FOR;
//
//		IF gDriver.TR[i].Cmd[C_TR_RESET] OR gDriver.ResetAll THEN
//			gDriver.TR[i].Cmd[C_TR_RESET] := FALSE;
//			brsmemset(ADR(gDriver.TR[i].Mon),0,SIZEOF(gDriver.TR[i].Mon));
//			brsmemset(ADR(gDriver.TR[i].Cmd),0,SIZEOF(gDriver.TR[i].Cmd));
//			brsmemset(ADR(gDriver.TR[i].Sev),0,SIZEOF(gDriver.TR[i].Sev));
//			brsmemset(ADR(gDriver.TR[i].Status),0,SIZEOF(gDriver.TR[i].Status));
//		END_IF;
//		IF gDriver.TR[i].Cmd[C_TR_CLEARCMD] THEN
//			gDriver.TR[i].Cmd[C_TR_CLEARCMD] := FALSE;
//			brsmemset(ADR(gDriver.TR[i].Cmd),0,SIZEOF(gDriver.TR[i].Cmd));
//		END_IF;
//		IF gDriver.TR[i].Cmd[C_TR_CLEARMON] THEN
//			gDriver.TR[i].Cmd[C_TR_CLEARMON] := FALSE;
//			brsmemset(ADR(gDriver.TR[i].Status.Severity),0,SIZEOF(gDriver.TR[i].Status.Severity));
//			brsmemset(ADR(gDriver.TR[i].Sev),0,SIZEOF(gDriver.TR[i].Sev));
//			brsmemset(ADR(gDriver.TR[i].Par.Mon),0,SIZEOF(gDriver.TR[i].Par.Mon));
//		END_IF;
//		IF gDriver.TR[i].Cmd[C_TR_DEFAULTMON] THEN
//			gDriver.TR[i].Cmd[C_TR_DEFAULTMON] := FALSE;
//			brsmemcpy(ADR(gDriver.TR[i].Par.Mon),ADR(gDriver.TR[i].DefaultPar.Mon),SIZEOF(gDriver.TR[i].Par.Mon));
//		END_IF;
//		IF gDriver.TR[i].Cmd[C_TR_CLEARPAR] THEN
//			gDriver.TR[i].Cmd[C_TR_CLEARPAR] := FALSE;
//			brsmemset(ADR(gDriver.TR[i].Par),0,SIZEOF(gDriver.TR[i].Par));
//		END_IF;
//		IF gDriver.TR[i].Cmd[C_TR_DEFAULTPAR] THEN
//			gDriver.TR[i].Cmd[C_TR_DEFAULTPAR] := FALSE;
//			brsmemcpy(ADR(gDriver.TR[i].Par),ADR(gDriver.TR[i].DefaultPar),SIZEOF(gDriver.TR[i].Par));
//		END_IF;
//		IF gDriver.TR[i].Cmd[C_TR_SAVEPAR] THEN
//			gDriver.TR[i].Cmd[C_TR_SAVEPAR] := FALSE;
//			brsmemcpy(ADR(gPar.Driver.TR[i]),ADR(gDriver.TR[i].Par),SIZEOF(gDriver.TR[i].Par));
//		END_IF;
//		IF gDriver.TR[i].Cmd[C_TR_LOADPAR] THEN
//			gDriver.TR[i].Cmd[C_TR_LOADPAR] := FALSE;
//			brsmemcpy(ADR(gDriver.TR[i].Par),ADR(gPar.Driver.TR[i]),SIZEOF(gDriver.TR[i].Par));
//		END_IF;
//
////
//// Implementation
////
//	    gDriver.TR[i].Status.McPathGenCusMechDir.Input.JointPos := gDriver.CN[i].Status.Position_mcJACS;
//	    gDriver.TR[i].Status.McPathGenCusMechDir.Input.TcpRefPos := gDriver.TR[i].Status.McPathGenCusMechDir.Output.TcpPos;
//	    gDriver.TR[i].Status.McPathGenCusMechDir.Parameter.CustomDataAddr := ADR(gDriver.TR[i].Status.CusMechData);
//	    gDriver.TR[i].Status.McPathGenCusMechDir.Parameter.JointCount := MAX_AXIS_V_IDX+1;
//	    customDirect(gDriver.TR[i].Status.McPathGenCusMechDir);
//
//		IF gDriver.TR[i].Cmd[C_TR_ENABLE] THEN
//			IF NOT gDriver.TR[i].Status.Active THEN
//				gDriver.TR[i].Status.TcpSetpoint := gDriver.TR[i].Status.McPathGenCusMechDir.Output.TcpPos;
//				gDriver.TR[i].Status.TcpSetpointLastStable := gDriver.TR[i].Status.McPathGenCusMechDir.Output.TcpPos;
//				brsmemset(ADR(gDriver.TR[i].Status.VelCmd),0,SIZEOF(gDriver.TR[i].Status.VelCmd));
//			ELSE
//				FOR j := 0 TO 14 DO
//					IF j <=2 THEN
//						IF gDriver.TR[i].Par.ControlMode = TR_CONTROL_MODE_COORD OR gDriver.TR[i].Par.ControlMode = TR_CONTROL_MODE_TRANS THEN
//							gDriver.TR[i].Status.LimitedCmd[j] := gDriver.TR[i].Status.InputCmd[j]*gDriver.TR[i].Par.VelocityFactor*20.0;
//						ELSE
//							gDriver.TR[i].Status.LimitedCmd[j] := 0.0;
//						END_IF;
//					ELSE
//						IF gDriver.TR[i].Par.ControlMode = TR_CONTROL_MODE_COORD OR gDriver.TR[i].Par.ControlMode = TR_CONTROL_MODE_ROTATE THEN
//							gDriver.TR[i].Status.LimitedCmd[j] := gDriver.TR[i].Status.InputCmd[j]*gDriver.TR[i].Par.VelocityFactor;
//						ELSE
//							gDriver.TR[i].Status.LimitedCmd[j] := 0.0;
//						END_IF;
//					END_IF;
//					IF gDriver.TR[i].Status.MTBasicsPID_0[j].PIDParameters.Gain <> gDriver.TR[i].Par.Gain THEN
//						gDriver.TR[i].Status.MTBasicsPID_0[j].PIDParameters.Gain := gDriver.TR[i].Par.Gain;
//						gDriver.TR[i].Status.MTBasicsPID_0[j].Update := TRUE;
//					END_IF;
//					IF gDriver.TR[i].Status.MTBasicsPID_0[j].PIDParameters.IntegrationTime <> gDriver.TR[i].Par.IntegralTime THEN
//						gDriver.TR[i].Status.MTBasicsPID_0[j].PIDParameters.IntegrationTime := gDriver.TR[i].Par.IntegralTime;
//						gDriver.TR[i].Status.MTBasicsPID_0[j].Update := TRUE;
//					END_IF;
//					gDriver.TR[i].Status.MTBasicsPID_0[j](Enable := TRUE, SetValue := 0.05, ActValue := ABS(LREAL_TO_REAL(gDriver.TR[i].Status.Lag[j])), MinOut := -0.999, MaxOut := 0.0);
//					gDriver.TR[i].Status.MTBasicsPID_0[j].Update := FALSE;
//					gDriver.TR[i].Status.Override := 1.0;
//					FOR k := 0 TO 14 DO
//						IF gDriver.TR[i].Status.Override > (1.0+gDriver.TR[i].Status.MTBasicsPID_0[k].Out) THEN
//							gDriver.TR[i].Status.Override := (1.0+gDriver.TR[i].Status.MTBasicsPID_0[k].Out);
//						END_IF;
//					END_FOR;
//					gDriver.TR[i].Status.LimitedCmd[j] := gDriver.TR[i].Status.LimitedCmd[j]*gDriver.TR[i].Status.Override;
//					gDriver.TR[i].Status.VelCmd[j] := gDriver.TR[i].Par.Filter*gDriver.TR[i].Status.VelCmd[j] + (1.0-gDriver.TR[i].Par.Filter)*gDriver.TR[i].Status.LimitedCmd[j];
//				END_FOR;
//				IF gDriver.TR[i].Par.WorldCoordMode THEN
//				    gDriver.TR[i].Status.VelCmd_World := gDriver.TR[i].Status.VelCmd;
//				ELSE
//	    			BuildTransform(gDriver.TR[i].Status.TcpSetpoint[0], gDriver.TR[i].Status.TcpSetpoint[1], gDriver.TR[i].Status.TcpSetpoint[2], gDriver.TR[i].Status.TcpSetpoint[3], gDriver.TR[i].Status.TcpSetpoint[4], gDriver.TR[i].Status.TcpSetpoint[5], ADR(gDriver.TR[i].Status.TcpMatrix));
//				    gDriver.TR[i].Status.VelCmd_World[0] := gDriver.TR[i].Status.TcpMatrix[0,0]*gDriver.TR[i].Status.VelCmd[0] + gDriver.TR[i].Status.TcpMatrix[0,1]*gDriver.TR[i].Status.VelCmd[1] + gDriver.TR[i].Status.TcpMatrix[0,2]*gDriver.TR[i].Status.VelCmd[2];
//				    gDriver.TR[i].Status.VelCmd_World[1] := gDriver.TR[i].Status.TcpMatrix[1,0]*gDriver.TR[i].Status.VelCmd[0] + gDriver.TR[i].Status.TcpMatrix[1,1]*gDriver.TR[i].Status.VelCmd[1] + gDriver.TR[i].Status.TcpMatrix[1,2]*gDriver.TR[i].Status.VelCmd[2];
//				    gDriver.TR[i].Status.VelCmd_World[2] := gDriver.TR[i].Status.TcpMatrix[2,0]*gDriver.TR[i].Status.VelCmd[0] + gDriver.TR[i].Status.TcpMatrix[2,1]*gDriver.TR[i].Status.VelCmd[1] + gDriver.TR[i].Status.TcpMatrix[2,2]*gDriver.TR[i].Status.VelCmd[2];
//				    gDriver.TR[i].Status.VelCmd_World[3] := gDriver.TR[i].Status.TcpMatrix[0,0]*gDriver.TR[i].Status.VelCmd[3] + gDriver.TR[i].Status.TcpMatrix[0,1]*gDriver.TR[i].Status.VelCmd[4] + gDriver.TR[i].Status.TcpMatrix[0,2]*gDriver.TR[i].Status.VelCmd[5];
//				    gDriver.TR[i].Status.VelCmd_World[4] := gDriver.TR[i].Status.TcpMatrix[1,0]*gDriver.TR[i].Status.VelCmd[3] + gDriver.TR[i].Status.TcpMatrix[1,1]*gDriver.TR[i].Status.VelCmd[4] + gDriver.TR[i].Status.TcpMatrix[1,2]*gDriver.TR[i].Status.VelCmd[5];
//				    gDriver.TR[i].Status.VelCmd_World[5] := gDriver.TR[i].Status.TcpMatrix[2,0]*gDriver.TR[i].Status.VelCmd[3] + gDriver.TR[i].Status.TcpMatrix[2,1]*gDriver.TR[i].Status.VelCmd[4] + gDriver.TR[i].Status.TcpMatrix[2,2]*gDriver.TR[i].Status.VelCmd[5];
//				END_IF;
//
//			    FOR j := 0 TO 14 DO
//			        IF gDriver.TR[i].Status.InverseStatus <> mcPATHGEN_CUSMECH_ERROR THEN
//			            gDriver.TR[i].Status.TcpSetpoint[j] := gDriver.TR[i].Status.TcpSetpoint[j] + gDriver.TR[i].Status.VelCmd_World[j];
//			        ELSE
//			            gDriver.TR[i].Status.TcpSetpoint[j] := gDriver.TR[i].Status.TcpSetpointLastStable[j] + gDriver.TR[i].Status.VelCmd_World[j];
//			        END_IF;
//			    END_FOR;
//			    gDriver.TR[i].Status.McPathGenCusMechInv.Parameter.CustomDataAddr := ADR(gDriver.TR[i].Status.CusMechData);
//			    gDriver.TR[i].Status.McPathGenCusMechInv.Input.JointRefPos := gDriver.TR[i].Status.McPathGenCusMechDir.Input.JointPos;
//			    gDriver.TR[i].Status.McPathGenCusMechInv.Parameter.JointCount := MAX_AXIS_V_IDX+1;
//			    gDriver.TR[i].Status.McPathGenCusMechInv.Input.TcpPos := gDriver.TR[i].Status.TcpSetpoint;
//			    gDriver.TR[i].Status.InverseStatus := customInverse(gDriver.TR[i].Status.McPathGenCusMechInv);
//			    IF gDriver.TR[i].Status.InverseStatus <> mcPATHGEN_CUSMECH_ERROR THEN
//					gDriver.TR[i].Status.TcpSetpointLastStable := gDriver.TR[i].Status.TcpSetpoint;
//			        gDriver.TR[i].Status.SetTCP := gDriver.TR[i].Status.McPathGenCusMechInv.Input.TcpPos;
//			        gDriver.TR[i].Status.SetJoint := gDriver.TR[i].Status.McPathGenCusMechInv.Output.JointPos;
//			    	gDriver.TR[i].Status.TotalLag := 0.0;
//					FOR j := 0 TO 14 DO
//			        	gDriver.TR[i].Status.Lag[j] := gDriver.TR[i].Status.SetJoint[j]-gDriver.TR[i].Status.McPathGenCusMechDir.Input.JointPos[j];
//			    		gDriver.TR[i].Status.TotalLag := gDriver.TR[i].Status.TotalLag + ABS(gDriver.TR[i].Status.Lag[j]);
//					END_FOR;
//			    END_IF;
//			END_IF;
//			gDriver.TR[i].Status.Active := TRUE;
//		ELSE
//			brsmemset(ADR(gDriver.TR[i].Status),0,SIZEOF(gDriver.TR[i].Status));
//		END_IF;
//
//		gDriver.TR[i].Wait[W_TR_NOERROR] := BOOL_TO_DINT(gDriver.TR[i].Status.InverseStatus <> mcPATHGEN_CUSMECH_ERROR);
//		gDriver.TR[i].Mon[M_TR_ERROR] := gDriver.TR[i].Status.InverseStatus = mcPATHGEN_CUSMECH_ERROR;
//	END_FOR;

END_ACTION
```

#### OMD_AB.st
```iecst
ACTION OMD_AB:

	gDriver.AB[DRIVER_INST_AB_VX_0].MpLinkADR 													:= ADR(gAxisVX_0);
	gDriver.AB[DRIVER_INST_AB_VY_0].MpLinkADR 													:= ADR(gAxisVY_0);
	gDriver.AB[DRIVER_INST_AB_VZ_0].MpLinkADR 													:= ADR(gAxisVZ_0);
	gDriver.AB[DRIVER_INST_AB_VT_0].MpLinkADR 													:= ADR(gAxisVT_0);
	gDriver.AB[DRIVER_INST_AB_VV_0].MpLinkADR 													:= ADR(gAxisVV_0);
	gDriver.AB[DRIVER_INST_AB_RX_0_0].MpLinkADR 												:= ADR(gAxisRX_0_0);
	gDriver.AB[DRIVER_INST_AB_RY_0_0].MpLinkADR 												:= ADR(gAxisRY_0_0);
	gDriver.AB[DRIVER_INST_AB_RZ_0_0].MpLinkADR 												:= ADR(gAxisRZ_0_0);
	gDriver.AB[DRIVER_INST_AB_RT_0_0].MpLinkADR 												:= ADR(gAxisRT_0_0);
	gDriver.AB[DRIVER_INST_AB_RV_0_0].MpLinkADR 												:= ADR(gAxisRV_0_0);
	gDriver.AB[DRIVER_INST_AB_RP_0_0].MpLinkADR 												:= ADR(gAxisRP_0_0);
	gDriver.AB[DRIVER_INST_AB_RP_1_0].MpLinkADR 												:= ADR(gAxisRP_1_0);

	FOR i := 0 TO MAX_DRIVER_AB_IDX DO
		IF NOT gDriver.AB[i].FirstScanComplete THEN
			gDriver.AB[i].FirstScanComplete 													:= TRUE;
			gDriver.AB[i].DefaultPar.AB.Acceleration											:= 50.0;							//RR
			gDriver.AB[i].DefaultPar.AB.AutoTune.FeedForward.Acceleration						:= 50.0;							//RR
			gDriver.AB[i].DefaultPar.AB.AutoTune.FeedForward.Direction							:= mcDIR_BOTH;						//McDirectionEnum
			gDriver.AB[i].DefaultPar.AB.AutoTune.FeedForward.MaxVelocityPercent					:= 50.0;							//RR
			gDriver.AB[i].DefaultPar.AB.AutoTune.FeedForward.Mode								:= mcACPAX_TUNE_FF_MODE_STANDARD; 	//McAcpAxAutoTuneFeedFwdModeEnum
			gDriver.AB[i].DefaultPar.AB.AutoTune.LoopFilterMode									:= mcAXIS_TUNE_LOOP_FILTER_F1;		//MpAxisAutoTuneLoopFilterModeEnum
			gDriver.AB[i].DefaultPar.AB.AutoTune.MaxCurrentPercent								:= 80.0;							//RR
			gDriver.AB[i].DefaultPar.AB.AutoTune.MaxDistance									:= 0.0;								//LR
			gDriver.AB[i].DefaultPar.AB.AutoTune.MaxPositionError								:= 1.0;								//LR
			gDriver.AB[i].DefaultPar.AB.AutoTune.Mode											:= mcAXIS_TUNE_AUTOMATIC;			//MpAxisAutoTuneModeEnum
			gDriver.AB[i].DefaultPar.AB.AutoTune.Options.MaxProportionalGain					:= 0.0;								//RR
			gDriver.AB[i].DefaultPar.AB.AutoTune.Options.SpeedTuneFilterTmeMode					:= mcACPAX_FILTER_TIME_USE;			//McAcpAxFilterTimeModeEnum
			gDriver.AB[i].DefaultPar.AB.AutoTune.Options.SpeedTuneLoopFilter1Mode				:= mcACPAX_LOOP_FILTER_IGNORE;		//McAcpAxLoopFilterModeEnum
			gDriver.AB[i].DefaultPar.AB.AutoTune.Orientation									:= mcACPAX_ORIENTATION_HORIZONTAL;	//McAcpAxAutoTuneOrientationEnum
			gDriver.AB[i].DefaultPar.AB.AutoTune.SaveControllerSettings							:= FALSE;							//BO
			gDriver.AB[i].DefaultPar.AB.Deceleration											:= 50.0;							//RR
			gDriver.AB[i].DefaultPar.AB.Direction												:= mcDIR_SHORTEST_WAY;				//McDirectionEnum
			gDriver.AB[i].DefaultPar.AB.Distance												:= 0.0;								//LR
			gDriver.AB[i].DefaultPar.AB.Homing.Mode												:= mcHOMING_DIRECT;					//McHomingModeEnum
			gDriver.AB[i].DefaultPar.AB.Homing.Position											:= 0.0;								//RR
			gDriver.AB[i].DefaultPar.AB.Homing.Options.Acceleration								:= 50.0;							//RR
			gDriver.AB[i].DefaultPar.AB.Homing.Options.AdditionalTorqueLimit.NegativeDirection	:= 0.0;								//RR
			gDriver.AB[i].DefaultPar.AB.Homing.Options.AdditionalTorqueLimit.PositiveDirection	:= 0.0;								//RR
			gDriver.AB[i].DefaultPar.AB.Homing.Options.BlockDetectionPositionError				:= 0.0;								//RR
			gDriver.AB[i].DefaultPar.AB.Homing.Options.DisableRestorePositionOnEnable			:= mcSWITCH_OFF;					//McSwitchEnum
			gDriver.AB[i].DefaultPar.AB.Homing.Options.DriveSpecificHoming						:= mcSWITCH_OFF;					//McSwitchEnum
			gDriver.AB[i].DefaultPar.AB.Homing.Options.DriveSpecificHomingMode					:= 0;								//SS
			gDriver.AB[i].DefaultPar.AB.Homing.Options.HomingDirection							:= mcDIR_POSITIVE;					//McDirectionEnum
			gDriver.AB[i].DefaultPar.AB.Homing.Options.HomingVelocity							:= 5.0;								//RR
			gDriver.AB[i].DefaultPar.AB.Homing.Options.KeepDirection							:= mcSWITCH_OFF;					//McSwitchEnum
			gDriver.AB[i].DefaultPar.AB.Homing.Options.PositionErrorStopLimit					:= 0.0;								//RR
			gDriver.AB[i].DefaultPar.AB.Homing.Options.ReferencePulse							:= mcSWITCH_OFF;					//McSwitchEnum
			gDriver.AB[i].DefaultPar.AB.Homing.Options.ReferencePulseBlockingDistance			:= 0.0;								//RR
			gDriver.AB[i].DefaultPar.AB.Homing.Options.RestorePositionVariableAddress			:= 0;								//UD
			gDriver.AB[i].DefaultPar.AB.Homing.Options.SensorOffset								:= 0.0;								//LR
			gDriver.AB[i].DefaultPar.AB.Homing.Options.SensorOffsetDirection					:= mcDIR_POSITIVE;					//McDirectionEnum
			gDriver.AB[i].DefaultPar.AB.Homing.Options.StartDirection							:= mcDIR_POSITIVE;					//McDirectionEnum
			gDriver.AB[i].DefaultPar.AB.Homing.Options.StartVelocity							:= 1.0;								//RR
			gDriver.AB[i].DefaultPar.AB.Homing.Options.SwitchEdge								:= mcDIR_POSITIVE;					//McDirectionEnum
			gDriver.AB[i].DefaultPar.AB.Homing.Options.TorqueLimit								:= 0.1;								//RR
			gDriver.AB[i].DefaultPar.AB.Jerk													:= 0.0;								//RR
			gDriver.AB[i].DefaultPar.AB.Jog.Acceleration										:= 50.0;							//RR
			gDriver.AB[i].DefaultPar.AB.Jog.Deceleration										:= 50.0;							//RR
			gDriver.AB[i].DefaultPar.AB.Jog.Jerk												:= 0.0;								//RR
			gDriver.AB[i].DefaultPar.AB.Jog.LimitPosition.FirstPosition							:= 0.0;								//LR
			gDriver.AB[i].DefaultPar.AB.Jog.LimitPosition.LastPosition							:= 0.0;								//LR
			gDriver.AB[i].DefaultPar.AB.Jog.Velocity											:= 5.0;								//RR
			gDriver.AB[i].DefaultPar.AB.LimitLoad.Direction										:= mcDIR_CURRENT;					//McDirectionEnum
			gDriver.AB[i].DefaultPar.AB.LimitLoad.Load											:= 2.0;								//RR
			gDriver.AB[i].DefaultPar.AB.Position												:= 0.0;								//LR
			gDriver.AB[i].DefaultPar.AB.Stop.Deceleration										:= 50.0;							//RR
			gDriver.AB[i].DefaultPar.AB.Stop.Jerk												:= 0.0;								//RR
			gDriver.AB[i].DefaultPar.AB.Stop.StopAtPosition.Activate							:= FALSE;							//BO
			gDriver.AB[i].DefaultPar.AB.Stop.StopAtPosition.Deceleration						:= 0.0;								//RR
			gDriver.AB[i].DefaultPar.AB.Stop.StopAtPosition.Position							:= 0.0;								//LR
			gDriver.AB[i].DefaultPar.AB.Velocity												:= 5.0;								//RR
			brsmemcpy(ADR(gDriver.AB[i].Par),ADR(gDriver.AB[i].DefaultPar),SIZEOF(gDriver.AB[i].Par));
		ELSIF NOT gDriver.AB[i].ParametersLoaded AND gMain.Services.Recipes.Out.ParametersReady THEN
			gDriver.AB[i].ParametersLoaded := TRUE;
			brsmemcpy(ADR(gDriver.AB[i].Par),ADR(gPar.Driver.AB[i]),SIZEOF(gDriver.AB[i].Par));
		END_IF;

		brsmemset(ADR(gDriver.AB[i].Sev),0,SIZEOF(gDriver.AB[i].Sev));
		brsmemset(ADR(gDriver.AB[i].Status),0,SIZEOF(gDriver.AB[i].Status));
		FOR j := 0 TO MAX_DRIVER_AB_MON_IDX DO
			IF gDriver.AB[i].Par.Mon[j].Enable THEN
				IF gDriver.AB[i].Mon[j] THEN
					gDriver.AB[i].CTON_Mon[j](IN := TRUE, PT := LREAL_TO_TIME(gDriver.AB[i].Par.Mon[j].Time*1000.0));
					IF gDriver.AB[i].CTON_Mon[j].Q THEN
						gDriver.AB[i].Sev[j] := gDriver.AB[i].Par.Mon[j].Sev;
						IF gDriver.AB[i].Status.Severity < gDriver.AB[i].Sev[j] THEN
							gDriver.AB[i].Status.Severity := gDriver.AB[i].Sev[j];
						END_IF;
					END_IF;
				ELSE
					gDriver.AB[i].CTON_Mon[j](IN := FALSE);
					gDriver.AB[i].Sev[j] := 0;
				END_IF;
			ELSE
				gDriver.AB[i].CTON_Mon[j](IN := FALSE);
				gDriver.AB[i].Sev[j] := 0;
			END_IF;
		END_FOR;
		IF gDriver.AB[i].Cmd[C_AB_RESET] OR gDriver.ResetAll THEN
			gDriver.AB[i].Cmd[C_AB_RESET] := FALSE;
			brsmemset(ADR(gDriver.AB[i].Mon),0,SIZEOF(gDriver.AB[i].Mon));
			brsmemset(ADR(gDriver.AB[i].Cmd),0,SIZEOF(gDriver.AB[i].Cmd));
			brsmemset(ADR(gDriver.AB[i].Sev),0,SIZEOF(gDriver.AB[i].Sev));
			brsmemset(ADR(gDriver.AB[i].Status),0,SIZEOF(gDriver.AB[i].Status));
		END_IF;
		IF gDriver.AB[i].Cmd[C_AB_CLEARCMD] THEN
			gDriver.AB[i].Cmd[C_AB_CLEARCMD] := FALSE;
			brsmemset(ADR(gDriver.AB[i].Cmd),0,SIZEOF(gDriver.AB[i].Cmd));
		END_IF;
		IF gDriver.AB[i].Cmd[C_AB_CLEARMON] THEN
			gDriver.AB[i].Cmd[C_AB_CLEARMON] := FALSE;
			brsmemset(ADR(gDriver.AB[i].Status.Severity),0,SIZEOF(gDriver.AB[i].Status.Severity));
			brsmemset(ADR(gDriver.AB[i].Sev),0,SIZEOF(gDriver.AB[i].Sev));
			brsmemset(ADR(gDriver.AB[i].Par.Mon),0,SIZEOF(gDriver.AB[i].Par.Mon));
		END_IF;
		IF gDriver.AB[i].Cmd[C_AB_DEFAULTMON] THEN
			gDriver.AB[i].Cmd[C_AB_DEFAULTMON] := FALSE;
			brsmemcpy(ADR(gDriver.AB[i].Par.Mon),ADR(gDriver.AB[i].DefaultPar.Mon),SIZEOF(gDriver.AB[i].Par.Mon));
		END_IF;
		IF gDriver.AB[i].Cmd[C_AB_CLEARPAR] THEN
			gDriver.AB[i].Cmd[C_AB_CLEARPAR] := FALSE;
			brsmemset(ADR(gDriver.AB[i].Par),0,SIZEOF(gDriver.AB[i].Par));
		END_IF;
		IF gDriver.AB[i].Cmd[C_AB_DEFAULTPAR] THEN
			gDriver.AB[i].Cmd[C_AB_DEFAULTPAR] := FALSE;
			brsmemcpy(ADR(gDriver.AB[i].Par),ADR(gDriver.AB[i].DefaultPar),SIZEOF(gDriver.AB[i].Par));
		END_IF;
		IF gDriver.AB[i].Cmd[C_AB_SAVEPAR] THEN
			gDriver.AB[i].Cmd[C_AB_SAVEPAR] := FALSE;
			brsmemcpy(ADR(gPar.Driver.AB[i]),ADR(gDriver.AB[i].Par),SIZEOF(gDriver.AB[i].Par));
		END_IF;
		IF gDriver.AB[i].Cmd[C_AB_LOADPAR] THEN
			gDriver.AB[i].Cmd[C_AB_LOADPAR] := FALSE;
			brsmemcpy(ADR(gDriver.AB[i].Par),ADR(gPar.Driver.AB[i]),SIZEOF(gDriver.AB[i].Par));
		END_IF;

		gDriver.AB[i].MpAxisBasic_0.ErrorReset			:= gDriver.AB[i].Cmd[C_AB_ERRORRESET] OR gMain.ErrorReset;
		gDriver.AB[i].MpAxisBasic_0.Home				:= gDriver.AB[i].Cmd[C_AB_HOME];
		gDriver.AB[i].MpAxisBasic_0.Power				:= gDriver.AB[i].Cmd[C_AB_POWER];
		gDriver.AB[i].MpAxisBasic_0.Update				:= gDriver.AB[i].Cmd[C_AB_UPDATE];
		gDriver.AB[i].MpAxisBasic_0.AutoTune			:= gDriver.AB[i].Cmd[C_AB_AUTOTUNE];
		gDriver.AB[i].MpAxisBasic_0.JogPositive			:= gDriver.AB[i].Cmd[C_AB_JOGPOSITIVE];
		gDriver.AB[i].MpAxisBasic_0.JogNegative			:= gDriver.AB[i].Cmd[C_AB_JOGNEGATIVE];
		gDriver.AB[i].MpAxisBasic_0.LimitLoad			:= gDriver.AB[i].Cmd[C_AB_LIMITLOAD];
		gDriver.AB[i].MpAxisBasic_0.Stop				:= gDriver.AB[i].Cmd[C_AB_STOP];
		gDriver.AB[i].MpAxisBasic_0.MoveAbsolute		:= gDriver.AB[i].Cmd[C_AB_MOVEABSOLUTE];
		gDriver.AB[i].MpAxisBasic_0.MoveAdditive		:= gDriver.AB[i].Cmd[C_AB_MOVEADDITIVE];
		gDriver.AB[i].MpAxisBasic_0.MoveVelocity		:= gDriver.AB[i].Cmd[C_AB_MOVEVELOCITY];
		gDriver.AB[i].MpAxisBasic_0.ReleaseBrake		:= gDriver.AB[i].Cmd[C_AB_RELEASEBRAKE];
		gDriver.AB[i].MpAxisBasic_0.Simulate			:= gDriver.AB[i].Cmd[C_AB_SIMULATE];

		gDriver.AB[i].MpAxisBasic_0(MpLink := gDriver.AB[i].MpLinkADR, Enable := TRUE, Parameters := ADR(gDriver.AB[i].Par.AB));

		gDriver.AB[i].Status.Position					:= gDriver.AB[i].MpAxisBasic_0.Position;
		gDriver.AB[i].Status.Velocity					:= gDriver.AB[i].MpAxisBasic_0.Velocity;

		gDriver.AB[i].Wait[W_AB_NOERROR]				:= BOOL_TO_DINT(NOT gDriver.AB[i].MpAxisBasic_0.Error);
		gDriver.AB[i].Wait[W_AB_COMMUNICATIONREADY]		:= BOOL_TO_DINT(gDriver.AB[i].MpAxisBasic_0.Info.CommunicationReady);
		gDriver.AB[i].Wait[W_AB_READYTOPOWERON]			:= BOOL_TO_DINT(gDriver.AB[i].MpAxisBasic_0.Info.ReadyToPowerOn);
		gDriver.AB[i].Wait[W_AB_POWERON]				:= BOOL_TO_DINT(gDriver.AB[i].MpAxisBasic_0.PowerOn);
		gDriver.AB[i].Wait[W_AB_ISHOMED]				:= BOOL_TO_DINT(gDriver.AB[i].MpAxisBasic_0.IsHomed AND NOT gDriver.AB[i].MpAxisBasic_0.CommandBusy);
		gDriver.AB[i].Wait[W_AB_LIMITLOADACTIVE]		:= BOOL_TO_DINT(gDriver.AB[i].MpAxisBasic_0.LimitLoadReady);
		gDriver.AB[i].Wait[W_AB_MOVEDONE]				:= BOOL_TO_DINT(gDriver.AB[i].MpAxisBasic_0.MoveDone);
		gDriver.AB[i].Wait[W_AB_UPDATEDONE]				:= BOOL_TO_DINT(gDriver.AB[i].MpAxisBasic_0.UpdateDone);
		gDriver.AB[i].Wait[W_AB_AUTOTUNEDONE]			:= BOOL_TO_DINT(gDriver.AB[i].MpAxisBasic_0.AutoTuneDone);
		gDriver.AB[i].Wait[W_AB_BRAKERELEASED]			:= BOOL_TO_DINT(gDriver.AB[i].MpAxisBasic_0.BrakeReleased);
		gDriver.AB[i].Wait[W_AB_COMMANDABORTED]			:= BOOL_TO_DINT(gDriver.AB[i].MpAxisBasic_0.CommandAborted);
		gDriver.AB[i].Wait[W_AB_COMMANDBUSY]			:= BOOL_TO_DINT(gDriver.AB[i].MpAxisBasic_0.CommandBusy);
		gDriver.AB[i].Wait[W_AB_INPOSITION]				:= BOOL_TO_DINT(gDriver.AB[i].MpAxisBasic_0.InPosition);
		gDriver.AB[i].Wait[W_AB_INVELOCITY]				:= BOOL_TO_DINT(gDriver.AB[i].MpAxisBasic_0.InVelocity);
		gDriver.AB[i].Wait[W_AB_MOVEACTIVE]				:= BOOL_TO_DINT(gDriver.AB[i].MpAxisBasic_0.MoveActive);
		gDriver.AB[i].Wait[W_AB_STOPPED]				:= BOOL_TO_DINT(gDriver.AB[i].MpAxisBasic_0.Stopped);
		gDriver.AB[i].Wait[W_AB_JOGGING]				:= BOOL_TO_DINT(gDriver.AB[i].MpAxisBasic_0.Info.Jogging);
		gDriver.AB[i].Wait[W_AB_JOGLIMITREACHED]		:= BOOL_TO_DINT(gDriver.AB[i].MpAxisBasic_0.Info.JogLimitReached);
		gDriver.AB[i].Wait[W_AB_SIMULATION]				:= BOOL_TO_DINT(gDriver.AB[i].MpAxisBasic_0.Info.Simulation);

		gDriver.AB[i].Mon[M_AB_ERROR]					:= gDriver.AB[i].MpAxisBasic_0.Error;
		gDriver.AB[i].Mon[M_AB_NOTPOWERON]				:= NOT gDriver.AB[i].MpAxisBasic_0.PowerOn;
	END_FOR;

//	McDirectionEnum :
//	(
//		mcDIR_POSITIVE := 0,							(*Movement only in the positive direction *)
//		mcDIR_NEGATIVE := 1,							(*Movement only in the negative direction*)
//		mcDIR_CURRENT := 2,								(*Movement in the direction of the active movement*)
//		mcDIR_SHORTEST_WAY := 3,						(*Movement with the shortest distance to the target, either in positive or negative direction. The movement will be in the positive direction if the distance is the same in both directions*)
//		mcDIR_EXCEED_PERIOD := 8,						(*The end position can be located outside of the axis period. The axis period can be exited in the negative direction if the end position is also negative*)
//		mcDIR_UNDEFINED := 9,							(*Movement in undefined direction*)
//		mcDIR_BOTH := 10								(*Movement in both directions*)
//	);
//	McSwitchEnum :
//	(
//		mcSWITCH_OFF := 0,		 						(*State/Behavior selection switched off*)
//		mcSWITCH_ON := 1			 					(*State/Behavior selection switched on*)
//	);
//	McHomingModeEnum :
//	(
//		mcHOMING_DIRECT := 0,							(*Direct homing. "Position" is used directly as the new axis position*)
//		mcHOMING_SWITCH_GATE := 1,						(*Homing with reference gate*)
//		mcHOMING_ABSOLUTE_SWITCH := 2,					(*Performs homing with absolute reference switch*)
//		mcHOMING_LIMIT_SWITCH := 4,	    				(*Homing with hardware limit switch*)
//		mcHOMING_ABSOLUTE := 5,							(*Homing by setting the "Position" homing offset for an absolute encoder*)
//		mcHOMING_DCM := 7,								(*Homing using interval-encoded reference marks*)
//		mcHOMING_BLOCK_TORQUE := 9,						(*Performs homing to mechanical limit, torque as criteria*)
//		mcHOMING_BLOCK_LAG_ERROR := 10,					(*Performs homing to mechanical limit, lag error as criteria*)
//		mcHOMING_ABSOLUTE_CORRECTION := 133,  			(*Homing by setting the "Position" homing offset for an absolute encoder with counter range correction. This mode must be used if the overflow of the absolute encoder is within the axis range of movement*)
//		mcHOMING_DCM_CORRECTION := 135,	 				(*Homing using distance-coded reference marks with counting range correction*)
//		mcHOMING_DEFAULT := 140,		 				(*All parameters, including "Position", are taken from the initial configuration for the axis*)
//		mcHOMING_INIT := 141,							(*All parameters, including "Position", are taken from an earlier initialization made using function block MC_BR_InitHome*)
//		mcHOMING_RESTORE_POSITION := 142				(*Restores position from a remanent variable*)
//	);
//	MpAxisAutoTuneModeEnum :
//	(
//		mcAXIS_TUNE_AUTOMATIC := 0, 					(* Performs a complete auto-tuning sequence of all controllers*)
//		mcAXIS_TUNE_SPEED := 1, 						(* Speed controller tuning*)
//		mcAXIS_TUNE_POSITION := 2, 						(* Position controller tuning*)
//		mcAXIS_TUNE_TEST := 3, 							(* Tests system stability*)
//		mcAXIS_TUNE_LOOP_FILTER := 4, 					(* Loop filter tuning*)
//		mcAXIS_TUNE_FEED_FORWARD := 5 					(*Feed forward tuning*)
//	);
//	MpAxisAutoTuneLoopFilterModeEnum :
//	(
//		mcAXIS_TUNE_LOOP_FILTER_F1 := 0, 				(*Tuning of loop filter 1 as a notch filter*)
//		mcAXIS_TUNE_LOOP_FILTER_F1_F2 := 1, 			(*Tuning of filter 1 and 2 as a notch filter*)
//		mcAXIS_TUNE_LOOP_FILTER_F1_F2_F3 := 2 			(*Tuning of filter 1, 2 and 3 as a notch filter*)
//	);
//	McAcpAxAutoTuneOrientationEnum:
//	(
//		mcACPAX_ORIENTATION_HORIZONTAL := 0, 		 	(*Horizontal orientation*)
//		mcACPAX_ORIENTATION_VERTICAL := 1    		 	(*Vertical orientation*)
//	);
//	McAcpAxFilterTimeModeEnum:
//	(
//		mcACPAX_FILTER_TIME_USE := 0,  					(*The determination of filter time constants is disabled; however, filter time constants are taken into account for autotuning*)
//		mcACPAX_FILTER_TIME_TUNE_MODE1 := 1, 		 	(*The controlled variable is the unfiltered actual speed n*)
//		mcACPAX_FILTER_TIME_TUNE_MODE2 := 2  		 	(*The controlled variable is the filtered actual speed n*)
//	);
//	McAcpAxLoopFilterModeEnum:
//	(
//		mcACPAX_LOOP_FILTER_IGNORE := 0,  				(*Loop filters are neither taken into account nor calculated.*)
//		mcACPAX_LOOP_FILTER_USE := 1,  					(*The parameters for all loop filters are taken into account for autotuning*)
//		mcACPAX_LOOP_FILTER_TUNE_NOTCH := 2  			(*The parameters for the loop filter are calculated*)
//	);
//	McAcpAxAutoTuneFeedFwdModeEnum:
//	(
//		mcACPAX_TUNE_FF_MODE_STANDARD := 0, 			(*Standard (active) tuning mode*)
//		mcACPAX_TUNE_FF_MODE_PASSIVE := 1 				(*Passive tuning mode*)
//	);
//	McAcpAxAutoTuneFeedFwdCmdEnum:
//	(
//		mcACPAX_TUNE_FF_CMD_START := 0, 				(*Start (standard or passive) tuning process*)
//		mcACPAX_TUNE_FF_CMD_FINISH := 1, 				(*Finish (passive) tuning process*)
//		mcACPAX_TUNE_FF_CMD_ABORT := 2 					(*Abort (stop) (passive) tuning process*)
//	);

END_ACTION
```

#### OMD_CS.st
```iecst
ACTION OMD_CS:

	gDriver.CS[DRIVER_INST_CS_VX_0].MpLinkADR 								:= ADR(gAxisVX_0);
	gDriver.CS[DRIVER_INST_CS_VX_0].CyclicPositionSetpoint[0]				:= gDriver.TR[0].Status.SetJoint[0];
	gDriver.CS[DRIVER_INST_CS_VX_0].CyclicVelocitySetpoint[0]				:= 0.0;
	gDriver.CS[DRIVER_INST_CS_VX_0].CyclicTorqueSetpoint[0]					:= 0.0;
	gDriver.CS[DRIVER_INST_CS_VX_0].CyclicTorqueFeedForwardSetpoint[0]		:= 0.0;

	gDriver.CS[DRIVER_INST_CS_VY_0].MpLinkADR 								:= ADR(gAxisVY_0);
	gDriver.CS[DRIVER_INST_CS_VY_0].CyclicPositionSetpoint[0]				:= gDriver.TR[0].Status.SetJoint[1];
	gDriver.CS[DRIVER_INST_CS_VY_0].CyclicVelocitySetpoint[0]				:= 0.0;
	gDriver.CS[DRIVER_INST_CS_VY_0].CyclicTorqueSetpoint[0]					:= 0.0;
	gDriver.CS[DRIVER_INST_CS_VY_0].CyclicTorqueFeedForwardSetpoint[0]		:= 0.0;

	gDriver.CS[DRIVER_INST_CS_VZ_0].MpLinkADR 								:= ADR(gAxisVZ_0);
	gDriver.CS[DRIVER_INST_CS_VZ_0].CyclicPositionSetpoint[0]				:= gDriver.TR[0].Status.SetJoint[2];
	gDriver.CS[DRIVER_INST_CS_VZ_0].CyclicVelocitySetpoint[0]				:= 0.0;
	gDriver.CS[DRIVER_INST_CS_VZ_0].CyclicTorqueSetpoint[0]					:= 0.0;
	gDriver.CS[DRIVER_INST_CS_VZ_0].CyclicTorqueFeedForwardSetpoint[0]		:= 0.0;

	gDriver.CS[DRIVER_INST_CS_VT_0].MpLinkADR 								:= ADR(gAxisVT_0);
	gDriver.CS[DRIVER_INST_CS_VT_0].CyclicPositionSetpoint[0]				:= gDriver.TR[0].Status.SetJoint[3];
	gDriver.CS[DRIVER_INST_CS_VT_0].CyclicVelocitySetpoint[0]				:= 0.0;
	gDriver.CS[DRIVER_INST_CS_VT_0].CyclicTorqueSetpoint[0]					:= 0.0;
	gDriver.CS[DRIVER_INST_CS_VT_0].CyclicTorqueFeedForwardSetpoint[0]		:= 0.0;

	gDriver.CS[DRIVER_INST_CS_VV_0].MpLinkADR 								:= ADR(gAxisVV_0);
	gDriver.CS[DRIVER_INST_CS_VV_0].CyclicPositionSetpoint[0]				:= gDriver.TR[0].Status.SetJoint[4];
	gDriver.CS[DRIVER_INST_CS_VV_0].CyclicVelocitySetpoint[0]				:= 0.0;
	gDriver.CS[DRIVER_INST_CS_VV_0].CyclicTorqueSetpoint[0]					:= 0.0;
	gDriver.CS[DRIVER_INST_CS_VV_0].CyclicTorqueFeedForwardSetpoint[0]		:= 0.0;

	gDriver.CS[DRIVER_INST_CS_RX_0_0].MpLinkADR 							:= ADR(gAxisRX_0_0);
	gDriver.CS[DRIVER_INST_CS_RX_0_0].CyclicPositionSetpoint[0]				:= gDriver.AB[DRIVER_INST_AB_VX_0].MpAxisBasic_0.Position;
	gDriver.CS[DRIVER_INST_CS_RX_0_0].CyclicVelocitySetpoint[0]				:= gDriver.AB[DRIVER_INST_AB_VX_0].MpAxisBasic_0.Velocity;
	gDriver.CS[DRIVER_INST_CS_RX_0_0].CyclicTorqueSetpoint[0]				:= 0.0;
	gDriver.CS[DRIVER_INST_CS_RX_0_0].CyclicTorqueFeedForwardSetpoint[0]	:= 0.0;

	gDriver.CS[DRIVER_INST_CS_RY_0_0].MpLinkADR 							:= ADR(gAxisRY_0_0);
	gDriver.CS[DRIVER_INST_CS_RY_0_0].CyclicPositionSetpoint[0]				:= gDriver.AB[DRIVER_INST_AB_VY_0].MpAxisBasic_0.Position;
	gDriver.CS[DRIVER_INST_CS_RY_0_0].CyclicVelocitySetpoint[0]				:= gDriver.AB[DRIVER_INST_AB_VY_0].MpAxisBasic_0.Velocity;
	gDriver.CS[DRIVER_INST_CS_RY_0_0].CyclicTorqueSetpoint[0]				:= 0.0;
	gDriver.CS[DRIVER_INST_CS_RY_0_0].CyclicTorqueFeedForwardSetpoint[0]	:= 0.0;

	gDriver.CS[DRIVER_INST_CS_RZ_0_0].MpLinkADR 							:= ADR(gAxisRZ_0_0);
	gDriver.CS[DRIVER_INST_CS_RZ_0_0].CyclicPositionSetpoint[0]				:= gDriver.AB[DRIVER_INST_AB_VZ_0].MpAxisBasic_0.Position;
	gDriver.CS[DRIVER_INST_CS_RZ_0_0].CyclicVelocitySetpoint[0]				:= gDriver.AB[DRIVER_INST_AB_VZ_0].MpAxisBasic_0.Velocity;
	gDriver.CS[DRIVER_INST_CS_RZ_0_0].CyclicTorqueSetpoint[0]				:= 0.0;
	gDriver.CS[DRIVER_INST_CS_RZ_0_0].CyclicTorqueFeedForwardSetpoint[0]	:= 0.0;

	gDriver.CS[DRIVER_INST_CS_RT_0_0].MpLinkADR 							:= ADR(gAxisRT_0_0);
	gDriver.CS[DRIVER_INST_CS_RT_0_0].CyclicPositionSetpoint[0]				:= gDriver.AB[DRIVER_INST_AB_VT_0].MpAxisBasic_0.Position;
	gDriver.CS[DRIVER_INST_CS_RT_0_0].CyclicVelocitySetpoint[0]				:= gDriver.AB[DRIVER_INST_AB_VT_0].MpAxisBasic_0.Velocity;
	gDriver.CS[DRIVER_INST_CS_RT_0_0].CyclicTorqueSetpoint[0]				:= 0.0;
	gDriver.CS[DRIVER_INST_CS_RT_0_0].CyclicTorqueFeedForwardSetpoint[0]	:= 0.0;

	gDriver.CS[DRIVER_INST_CS_RV_0_0].MpLinkADR 							:= ADR(gAxisRV_0_0);
	gDriver.CS[DRIVER_INST_CS_RV_0_0].CyclicPositionSetpoint[0]				:= gDriver.AB[DRIVER_INST_AB_VV_0].MpAxisBasic_0.Position;
	gDriver.CS[DRIVER_INST_CS_RV_0_0].CyclicVelocitySetpoint[0]				:= gDriver.AB[DRIVER_INST_AB_VV_0].MpAxisBasic_0.Velocity;
	gDriver.CS[DRIVER_INST_CS_RV_0_0].CyclicTorqueSetpoint[0]				:= 0.0;
	gDriver.CS[DRIVER_INST_CS_RV_0_0].CyclicTorqueFeedForwardSetpoint[0]	:= 0.0;

	FOR i := 0 TO MAX_DRIVER_CS_IDX DO
		IF NOT gDriver.CS[i].FirstScanComplete THEN
			gDriver.CS[i].FirstScanComplete 													:= TRUE;
			gDriver.CS[i].DefaultPar.CS.MoveCyclicPosition.Acceleration							:= 0.0;								//RR
			gDriver.CS[i].DefaultPar.CS.MoveCyclicPosition.AlternativeValueSource				:= mcALT_VALUE_NOT_USED;			//McAltValueSrcEnum
			gDriver.CS[i].DefaultPar.CS.MoveCyclicPosition.Deceleration							:= 0.0;								//RR
			gDriver.CS[i].DefaultPar.CS.MoveCyclicPosition.DisableJoltLimitation				:= mcSWITCH_OFF;					//McSwitchEnum
			gDriver.CS[i].DefaultPar.CS.MoveCyclicPosition.InterpolationMode					:= mcIPLM_DEFAULT;					//McIplModeEnum
			gDriver.CS[i].DefaultPar.CS.MoveCyclicPosition.Jerk									:= 0.0;								//RR
			gDriver.CS[i].DefaultPar.CS.MoveCyclicPosition.Velocity								:= 0.0;								//RR
			gDriver.CS[i].DefaultPar.CS.MoveCyclicVelocity.Acceleration							:= 0.0;								//RR
			gDriver.CS[i].DefaultPar.CS.MoveCyclicVelocity.AlternativeValueSource				:= mcALT_VALUE_NOT_USED;			//McAltValueSrcEnum
			gDriver.CS[i].DefaultPar.CS.MoveCyclicVelocity.Deceleration							:= 0.0;								//RR
			gDriver.CS[i].DefaultPar.CS.MoveCyclicVelocity.DisableJoltLimitation				:= mcSWITCH_OFF;					//McSwitchEnum
			gDriver.CS[i].DefaultPar.CS.MoveCyclicVelocity.InterpolationMode					:= mcIPLM_DEFAULT;					//McIplModeEnum
			gDriver.CS[i].DefaultPar.CS.MoveCyclicVelocity.Jerk									:= 0.0;								//RR
			gDriver.CS[i].DefaultPar.CS.MoveCyclicVelocity.Mode									:= mcAXIS_MCV_MODE_MOVE_CYC_VEL;	//MpAxisMoveCyclicVelocityModeEnum
			gDriver.CS[i].DefaultPar.CS.TorqueControl.Acceleration								:= 0.0;								//RR
			gDriver.CS[i].DefaultPar.CS.TorqueControl.CmdIndependentActivation					:= FALSE;							//BO
			gDriver.CS[i].DefaultPar.CS.TorqueControl.Jerk										:= 0.0;								//RR
			gDriver.CS[i].DefaultPar.CS.TorqueControl.MaximumVelocity							:= 0.0;								//RR
			gDriver.CS[i].DefaultPar.CS.TorqueControl.MinimumVelocity							:= 0.0;								//RR
			gDriver.CS[i].DefaultPar.CS.TorqueControl.Options.CorrectVelocityLimits				:= FALSE;							//BO
			gDriver.CS[i].DefaultPar.CS.TorqueControl.Options.NoHomingCheck						:= FALSE;							//BO
			gDriver.CS[i].DefaultPar.CS.TorqueControl.Options.StartAlternativeValueSource		:= mcALT_VALUE_NOT_USED;			//McAltValueSrcEnum
			gDriver.CS[i].DefaultPar.CS.TorqueControl.Options.TimeLimit							:= 0.0;								//RR
			gDriver.CS[i].DefaultPar.CS.TorqueControl.Options.TorqueAlternativeValueSource		:= mcALT_VALUE_NOT_USED;			//McAltValueSrcEnum
			gDriver.CS[i].DefaultPar.CS.TorqueControl.Options.UseTimeLimit						:= FALSE;							//BO
			gDriver.CS[i].DefaultPar.CS.TorqueControl.Options.UseVelocityLimits					:= FALSE;							//BO
			gDriver.CS[i].DefaultPar.CS.TorqueControl.TorqueRamp								:= 0.0;								//RR
			gDriver.CS[i].DefaultPar.CS.TorqueControl.TorqueResolution							:= 0.0;								//RR
			gDriver.CS[i].DefaultPar.CS.TorqueFeedForward.InterpolationMode						:= mcIPLM_DEFAULT;					//McIplModeEnum
			gDriver.CS[i].DefaultPar.CS.TorqueFeedForward.Options.DisableMode					:= mcDISABLE_DEFAULT;				//McDisableModeEnum
			gDriver.CS[i].DefaultPar.CyclicPositionSource										:= 0;								//SD
			gDriver.CS[i].DefaultPar.CyclicTorqueSource											:= 0;								//SD
			gDriver.CS[i].DefaultPar.CyclicTorqueFeedForwardSource								:= 0;								//SD
			gDriver.CS[i].DefaultPar.CyclicVelocitySource										:= 0;								//SD
			brsmemcpy(ADR(gDriver.CS[i].Par),ADR(gDriver.CS[i].DefaultPar),SIZEOF(gDriver.CS[i].Par));
		ELSIF NOT gDriver.CS[i].ParametersLoaded AND gMain.Services.Recipes.Out.ParametersReady THEN
			gDriver.CS[i].ParametersLoaded := TRUE;
			brsmemcpy(ADR(gDriver.CS[i].Par),ADR(gPar.Driver.CS[i]),SIZEOF(gDriver.CS[i].Par));
		END_IF;

		brsmemset(ADR(gDriver.CS[i].Sev),0,SIZEOF(gDriver.CS[i].Sev));
		brsmemset(ADR(gDriver.CS[i].Status),0,SIZEOF(gDriver.CS[i].Status));
		FOR j := 0 TO MAX_DRIVER_CS_MON_IDX DO
			IF gDriver.CS[i].Par.Mon[j].Enable THEN
				IF gDriver.CS[i].Mon[j] THEN
					gDriver.CS[i].CTON_Mon[j](IN := TRUE, PT := LREAL_TO_TIME(gDriver.CS[i].Par.Mon[j].Time*1000.0));
					IF gDriver.CS[i].CTON_Mon[j].Q THEN
						gDriver.CS[i].Sev[j] := gDriver.CS[i].Par.Mon[j].Sev;
						IF gDriver.CS[i].Status.Severity < gDriver.CS[i].Sev[j] THEN
							gDriver.CS[i].Status.Severity := gDriver.CS[i].Sev[j];
						END_IF;
					END_IF;
				ELSE
					gDriver.CS[i].CTON_Mon[j](IN := FALSE);
					gDriver.CS[i].Sev[j] := 0;
				END_IF;
			ELSE
				gDriver.CS[i].CTON_Mon[j](IN := FALSE);
				gDriver.CS[i].Sev[j] := 0;
			END_IF;
		END_FOR;
		IF gDriver.CS[i].Cmd[C_CS_RESET] OR gDriver.ResetAll THEN
			gDriver.CS[i].Cmd[C_CS_RESET] := FALSE;
			brsmemset(ADR(gDriver.CS[i].Mon),0,SIZEOF(gDriver.CS[i].Mon));
			brsmemset(ADR(gDriver.CS[i].Cmd),0,SIZEOF(gDriver.CS[i].Cmd));
			brsmemset(ADR(gDriver.CS[i].Sev),0,SIZEOF(gDriver.CS[i].Sev));
			brsmemset(ADR(gDriver.CS[i].Status),0,SIZEOF(gDriver.CS[i].Status));
		END_IF;
		IF gDriver.CS[i].Cmd[C_CS_CLEARCMD] THEN
			gDriver.CS[i].Cmd[C_CS_CLEARCMD] := FALSE;
			brsmemset(ADR(gDriver.CS[i].Cmd),0,SIZEOF(gDriver.CS[i].Cmd));
		END_IF;
		IF gDriver.CS[i].Cmd[C_CS_CLEARMON] THEN
			gDriver.CS[i].Cmd[C_CS_CLEARMON] := FALSE;
			brsmemset(ADR(gDriver.CS[i].Status.Severity),0,SIZEOF(gDriver.CS[i].Status.Severity));
			brsmemset(ADR(gDriver.CS[i].Sev),0,SIZEOF(gDriver.CS[i].Sev));
			brsmemset(ADR(gDriver.CS[i].Par.Mon),0,SIZEOF(gDriver.CS[i].Par.Mon));
		END_IF;
		IF gDriver.CS[i].Cmd[C_CS_DEFAULTMON] THEN
			gDriver.CS[i].Cmd[C_CS_DEFAULTMON] := FALSE;
			brsmemcpy(ADR(gDriver.CS[i].Par.Mon),ADR(gDriver.CS[i].DefaultPar.Mon),SIZEOF(gDriver.CS[i].Par.Mon));
		END_IF;
		IF gDriver.CS[i].Cmd[C_CS_CLEARPAR] THEN
			gDriver.CS[i].Cmd[C_CS_CLEARPAR] := FALSE;
			brsmemset(ADR(gDriver.CS[i].Par),0,SIZEOF(gDriver.CS[i].Par));
		END_IF;
		IF gDriver.CS[i].Cmd[C_CS_DEFAULTPAR] THEN
			gDriver.CS[i].Cmd[C_CS_DEFAULTPAR] := FALSE;
			brsmemcpy(ADR(gDriver.CS[i].Par),ADR(gDriver.CS[i].DefaultPar),SIZEOF(gDriver.CS[i].Par));
		END_IF;
		IF gDriver.CS[i].Cmd[C_CS_SAVEPAR] THEN
			gDriver.CS[i].Cmd[C_CS_SAVEPAR] := FALSE;
			brsmemcpy(ADR(gPar.Driver.CS[i]),ADR(gDriver.CS[i].Par),SIZEOF(gDriver.CS[i].Par));
		END_IF;
		IF gDriver.CS[i].Cmd[C_CS_LOADPAR] THEN
			gDriver.CS[i].Cmd[C_CS_LOADPAR] := FALSE;
			brsmemcpy(ADR(gDriver.CS[i].Par),ADR(gPar.Driver.CS[i]),SIZEOF(gDriver.CS[i].Par));
		END_IF;
		gDriver.CS[i].MpAxisCyclicSet_0.ErrorReset						:= gDriver.CS[i].Cmd[C_CS_ERRORRESET] OR gMain.ErrorReset;
		gDriver.CS[i].MpAxisCyclicSet_0.MoveCyclicPosition				:= gDriver.CS[i].Cmd[C_CS_MOVECYCLICPOSITION];
		gDriver.CS[i].MpAxisCyclicSet_0.MoveCyclicVelocity				:= gDriver.CS[i].Cmd[C_CS_MOVECYCLICVELOCITY];
		gDriver.CS[i].MpAxisCyclicSet_0.TorqueControl					:= gDriver.CS[i].Cmd[C_CS_TORQUECONTROL];
		gDriver.CS[i].MpAxisCyclicSet_0.TorqueFeedForward				:= gDriver.CS[i].Cmd[C_CS_TORQUEFEEDFORWARD];
		gDriver.CS[i].MpAxisCyclicSet_0.Update							:= gDriver.CS[i].Cmd[C_CS_UPDATE];

		gDriver.CS[i].MpAxisCyclicSet_0.CyclicPosition					:= 0.0;
		IF gDriver.CS[i].Par.CyclicPositionSource <= MAX_DRIVER_CS_SOURCE_IDX THEN
			gDriver.CS[i].MpAxisCyclicSet_0.CyclicPosition				:= gDriver.CS[i].CyclicPositionSetpoint[gDriver.CS[i].Par.CyclicPositionSource];
		END_IF;
		gDriver.CS[i].MpAxisCyclicSet_0.CyclicVelocity					:= 0.0;
		IF gDriver.CS[i].Par.CyclicVelocitySource <= MAX_DRIVER_CS_SOURCE_IDX THEN
			gDriver.CS[i].MpAxisCyclicSet_0.CyclicVelocity				:= gDriver.CS[i].CyclicVelocitySetpoint[gDriver.CS[i].Par.CyclicVelocitySource];
		END_IF;
		gDriver.CS[i].MpAxisCyclicSet_0.CyclicTorque					:= 0.0;
		IF gDriver.CS[i].Par.CyclicTorqueSource <= MAX_DRIVER_CS_SOURCE_IDX THEN
			gDriver.CS[i].MpAxisCyclicSet_0.CyclicTorque 				:= gDriver.CS[i].CyclicTorqueSetpoint[gDriver.CS[i].Par.CyclicTorqueSource];
		END_IF;
		gDriver.CS[i].MpAxisCyclicSet_0.CyclicTorqueFeedForward			:= 0.0;
		IF gDriver.CS[i].Par.CyclicTorqueFeedForwardSource <= MAX_DRIVER_CS_SOURCE_IDX THEN
			gDriver.CS[i].MpAxisCyclicSet_0.CyclicTorqueFeedForward		:= gDriver.CS[i].CyclicTorqueFeedForwardSetpoint[gDriver.CS[i].Par.CyclicTorqueFeedForwardSource];
		END_IF;

		gDriver.CS[i].MpAxisCyclicSet_0(MpLink := gDriver.CS[i].MpLinkADR, Enable := TRUE, Parameters := ADR(gDriver.CS[i].Par.CS));

		gDriver.CS[i].Wait[W_CS_NOERROR]								:= BOOL_TO_DINT(NOT gDriver.CS[i].MpAxisCyclicSet_0.Error);
		gDriver.CS[i].Wait[W_CS_COMMANDABORTED]							:= BOOL_TO_DINT(gDriver.CS[i].MpAxisCyclicSet_0.CommandAborted);
		gDriver.CS[i].Wait[W_CS_COMMANDBUSY]							:= BOOL_TO_DINT(gDriver.CS[i].MpAxisCyclicSet_0.CommandBusy);
		gDriver.CS[i].Wait[W_CS_UPDATEDONE]								:= BOOL_TO_DINT(gDriver.CS[i].MpAxisCyclicSet_0.UpdateDone);
		gDriver.CS[i].Wait[W_CS_MOVECYCLICPOSITIONACTIVE]				:= BOOL_TO_DINT(gDriver.CS[i].MpAxisCyclicSet_0.MoveCyclicPositionActive);
		gDriver.CS[i].Wait[W_CS_MOVECYCLICVELOCITYACTIVE]				:= BOOL_TO_DINT(gDriver.CS[i].MpAxisCyclicSet_0.MoveCyclicVelocityActive);
		gDriver.CS[i].Wait[W_CS_TORQUECONTROLACTIVE]					:= BOOL_TO_DINT(gDriver.CS[i].MpAxisCyclicSet_0.TorqueControlActive);
		gDriver.CS[i].Wait[W_CS_TORQUEFEEDFORWARDACTIVE]				:= BOOL_TO_DINT(gDriver.CS[i].MpAxisCyclicSet_0.TorqueFeedForwardActive);
		gDriver.CS[i].Wait[W_CS_TCAXISLIMITACTIVE]						:= BOOL_TO_DINT(gDriver.CS[i].MpAxisCyclicSet_0.Info.TorqueControl.AxisLimitActive);
		gDriver.CS[i].Wait[W_CS_TCDATAINITIALIZED]						:= BOOL_TO_DINT(gDriver.CS[i].MpAxisCyclicSet_0.Info.TorqueControl.DataInitialized);
		gDriver.CS[i].Wait[W_CS_TCINTORQUE]								:= BOOL_TO_DINT(gDriver.CS[i].MpAxisCyclicSet_0.Info.TorqueControl.InTorque);
		gDriver.CS[i].Wait[W_CS_TCREADY]								:= BOOL_TO_DINT(gDriver.CS[i].MpAxisCyclicSet_0.Info.TorqueControl.Ready);
		gDriver.CS[i].Wait[W_CS_AXISREADY]								:= BOOL_TO_DINT(gDriver.CS[i].MpAxisCyclicSet_0.Info.AxisReady);

		gDriver.CS[i].Mon[M_CS_ERROR]									:= gDriver.CS[i].MpAxisCyclicSet_0.Error;
		gDriver.CS[i].Mon[M_CS_NOTMOVECYCLICPOSITIONACTIVE]				:= NOT gDriver.CS[i].MpAxisCyclicSet_0.MoveCyclicPositionActive;
		gDriver.CS[i].Mon[M_CS_NOTMOVECYCLICVELOCITYACTIVE]				:= NOT gDriver.CS[i].MpAxisCyclicSet_0.MoveCyclicVelocityActive;
		gDriver.CS[i].Mon[M_CS_NOTTORQUECONTROLACTIVE]					:= NOT gDriver.CS[i].MpAxisCyclicSet_0.TorqueControlActive;
		gDriver.CS[i].Mon[M_CS_NOTTORQUEFEEDFORWARDACTIVE]				:= NOT gDriver.CS[i].MpAxisCyclicSet_0.TorqueFeedForwardActive;
		gDriver.CS[i].Mon[M_CS_TCAXISLIMITACTIVE]						:= gDriver.CS[i].MpAxisCyclicSet_0.Info.TorqueControl.AxisLimitActive;
		gDriver.CS[i].Mon[M_CS_NOTTCINTORQUE]							:= NOT gDriver.CS[i].MpAxisCyclicSet_0.Info.TorqueControl.InTorque;
	END_FOR;

//	MpAxisMoveCyclicVelocityModeEnum :
//	(
//		mcAXIS_MCV_MODE_MOVE_CYC_VEL, 	(*MoveCyclicVelocity mode*)
//		mcAXIS_MCV_MODE_MOVE_VEL_CTRL 	(*VelocityControl mode*)
//	);
//	McIplModeEnum :
//	(
//		mcIPLM_DEFAULT,					(*The most suitable available interpolation is used*)
//		mcIPLM_OFF,						(*Interpolation off*)
//		mcIPLM_LINEAR,					(*linear interpolation*)
//		mcIPLM_QUADRATIC,				(*quadratic interpolation*)
//		mcIPLM_QUADRATIC_NO_OVERSHOOT	(*quadratic interpolation without overshoot*)
//	);
//	McAltValueSrcEnum :
//	(
//		mcALT_VALUE_NOT_USED := 0,		(*No alternative value source is used*)
//		mcALT_VALUE1 := 1,				(*"Value source 1" of the feature "Alternative value source" is used*)
//		mcALT_VALUE2 := 2,				(*"Value source 2" of the feature "Alternative value source" is used*)
//		mcALT_VALUE3 := 3,				(*"Value source 3" of the feature "Alternative value source" is used*)
//		mcALT_VALUE4 := 4,				(*"Value source 4" of the feature "Alternative value source" is used*)
//		mcALT_VALUE5 := 5,				(*"Value source 5" of the feature "Alternative value source" is used*)
//		mcALT_VALUE6 := 6,				(*"Value source 6" of the feature "Alternative value source" is used*)
//		mcALT_VALUE7 := 7,				(*"Value source 7" of the feature "Alternative value source" is used*)
//		mcALT_VALUE8 := 8				(*"Value source 8" of the feature "Alternative value source" is used*)
//	);
//	McSwitchEnum :
//	(
//		mcSWITCH_OFF,					(*State/Behavior selection switched off*)
//		mcSWITCH_ON			 			(*State/Behavior selection switched on*)
//	);
//	McDisableModeEnum :
//	(
//		mcDISABLE_DEFAULT := 0, 		(*Switch to default setting at disable*)
//		mcDISABLE_KEEP_VALUE := 1 		(*Keep value at disable*)
//	);

END_ACTION
```

#### OMD_FI.st
```iecst
ACTION OMD_FI:

	//TESTING
	//gDriver.CS[DRIVER_INST_CS_RX0_0].Par.CyclicPosition := gDriver.AB[DRIVER_INST_AB_VX_0].MpAxisBasic_0.Position;
//	gDriver.CS[DRIVER_INST_CS_RX0_0].MpLinkADR 							:= ADR(gAxisRX0_0);
//	gDriver.CS[DRIVER_INST_CS_RX0_0].CyclicPositionSetpoint[0]			:= gDriver.AB[DRIVER_INST_AB_VX_0].MpAxisBasic_0.Position;
//	gDriver.CS[DRIVER_INST_CS_RX0_0].CyclicVelocitySetpoint[0]			:= gDriver.AB[DRIVER_INST_AB_VX_0].MpAxisBasic_0.Velocity;
//	gDriver.CS[DRIVER_INST_CS_RX0_0].CyclicTorqueSetpoint[0]			:= 0.0;
//	gDriver.CS[DRIVER_INST_CS_RX0_0].CyclicTorqueFeedForwardSetpoint[0]	:= 0.0;
//
//	gDriver.CS[DRIVER_INST_CS_RY0_0].MpLinkADR 							:= ADR(gAxisRY0_0);
//	gDriver.CS[DRIVER_INST_CS_RY0_0].CyclicPositionSetpoint[0]			:= gDriver.AB[DRIVER_INST_AB_VY_0].MpAxisBasic_0.Position;
//	gDriver.CS[DRIVER_INST_CS_RY0_0].CyclicVelocitySetpoint[0]			:= gDriver.AB[DRIVER_INST_AB_VY_0].MpAxisBasic_0.Velocity;
//	gDriver.CS[DRIVER_INST_CS_RY0_0].CyclicTorqueSetpoint[0]			:= 0.0;
//	gDriver.CS[DRIVER_INST_CS_RY0_0].CyclicTorqueFeedForwardSetpoint[0]	:= 0.0;
//
//	gDriver.CS[DRIVER_INST_CS_RZ0_0].MpLinkADR 							:= ADR(gAxisRZ0_0);
//	gDriver.CS[DRIVER_INST_CS_RZ0_0].CyclicPositionSetpoint[0]			:= gDriver.AB[DRIVER_INST_AB_VZ_0].MpAxisBasic_0.Position;
//	gDriver.CS[DRIVER_INST_CS_RZ0_0].CyclicVelocitySetpoint[0]			:= gDriver.AB[DRIVER_INST_AB_VZ_0].MpAxisBasic_0.Velocity;
//	gDriver.CS[DRIVER_INST_CS_RZ0_0].CyclicTorqueSetpoint[0]			:= 0.0;
//	gDriver.CS[DRIVER_INST_CS_RZ0_0].CyclicTorqueFeedForwardSetpoint[0]	:= 0.0;
//
//	gDriver.CS[DRIVER_INST_CS_RT0_0].MpLinkADR 							:= ADR(gAxisRT0_0);
//	gDriver.CS[DRIVER_INST_CS_RT0_0].CyclicPositionSetpoint[0]			:= gDriver.AB[DRIVER_INST_AB_VT_0].MpAxisBasic_0.Position;
//	gDriver.CS[DRIVER_INST_CS_RT0_0].CyclicVelocitySetpoint[0]			:= gDriver.AB[DRIVER_INST_AB_VT_0].MpAxisBasic_0.Velocity;
//	gDriver.CS[DRIVER_INST_CS_RT0_0].CyclicTorqueSetpoint[0]			:= 0.0;
//	gDriver.CS[DRIVER_INST_CS_RT0_0].CyclicTorqueFeedForwardSetpoint[0]	:= 0.0;
//
//	gDriver.CS[DRIVER_INST_CS_RV0_0].MpLinkADR 							:= ADR(gAxisRV0_0);
//	gDriver.CS[DRIVER_INST_CS_RV0_0].CyclicPositionSetpoint[0]			:= gDriver.AB[DRIVER_INST_AB_VV_0].MpAxisBasic_0.Position;
//	gDriver.CS[DRIVER_INST_CS_RV0_0].CyclicVelocitySetpoint[0]			:= gDriver.AB[DRIVER_INST_AB_VV_0].MpAxisBasic_0.Velocity;
//	gDriver.CS[DRIVER_INST_CS_RV0_0].CyclicTorqueSetpoint[0]			:= 0.0;
//	gDriver.CS[DRIVER_INST_CS_RV0_0].CyclicTorqueFeedForwardSetpoint[0]	:= 0.0;
//
//	FOR i := 0 TO MAX_DRIVER_CS_IDX DO
//		gDriver.CS[i].MpAxisCyclicSet_0.CyclicPosition					:= 0.0;
//		IF gDriver.CS[i].Par.CyclicPositionSource <= MAX_DRIVER_CS_SOURCE_IDX THEN
//			gDriver.CS[i].MpAxisCyclicSet_0.CyclicPosition				:= gDriver.CS[i].CyclicPositionSetpoint[gDriver.CS[i].Par.CyclicPositionSource];
//		END_IF;
//		gDriver.CS[i].MpAxisCyclicSet_0.CyclicVelocity					:= 0.0;
//		IF gDriver.CS[i].Par.CyclicVelocitySource <= MAX_DRIVER_CS_SOURCE_IDX THEN
//			gDriver.CS[i].MpAxisCyclicSet_0.CyclicVelocity				:= gDriver.CS[i].CyclicVelocitySetpoint[gDriver.CS[i].Par.CyclicVelocitySource];
//		END_IF;
//		gDriver.CS[i].MpAxisCyclicSet_0.CyclicTorque					:= 0.0;
//		IF gDriver.CS[i].Par.CyclicTorqueSource <= MAX_DRIVER_CS_SOURCE_IDX THEN
//			gDriver.CS[i].MpAxisCyclicSet_0.CyclicTorque 				:= gDriver.CS[i].CyclicTorqueSetpoint[gDriver.CS[i].Par.CyclicTorqueSource];
//		END_IF;
//		gDriver.CS[i].MpAxisCyclicSet_0.CyclicTorqueFeedForward			:= 0.0;
//		IF gDriver.CS[i].Par.CyclicTorqueFeedForwardSource <= MAX_DRIVER_CS_SOURCE_IDX THEN
//			gDriver.CS[i].MpAxisCyclicSet_0.CyclicTorqueFeedForward		:= gDriver.CS[i].CyclicTorqueFeedForwardSetpoint[gDriver.CS[i].Par.CyclicTorqueFeedForwardSource];
//		END_IF;
//
//		gDriver.CS[i].MpAxisCyclicSet_0.ErrorReset						:= gDriver.CS[i].Cmd[C_CS_ERRORRESET] OR gMain.ErrorReset;
//		gDriver.CS[i].MpAxisCyclicSet_0.MoveCyclicPosition				:= gDriver.CS[i].Cmd[C_CS_MOVECYCLICPOSITION];
//		gDriver.CS[i].MpAxisCyclicSet_0.MoveCyclicVelocity				:= gDriver.CS[i].Cmd[C_CS_MOVECYCLICVELOCITY];
//		gDriver.CS[i].MpAxisCyclicSet_0.TorqueControl					:= gDriver.CS[i].Cmd[C_CS_TORQUECONTROL];
//		gDriver.CS[i].MpAxisCyclicSet_0.TorqueFeedForward				:= gDriver.CS[i].Cmd[C_CS_TORQUEFEEDFORWARD];
//		gDriver.CS[i].MpAxisCyclicSet_0.Update							:= gDriver.CS[i].Cmd[C_CS_UPDATE];
//
//		gDriver.CS[i].MpAxisCyclicSet_0(MpLink := gDriver.CS[i].MpLinkADR, Enable := TRUE, Parameters := ADR(gDriver.CS[i].Par.CS));
//
//		gDriver.CS[i].Wait[W_CS_NOERROR]								:= BOOL_TO_DINT(NOT gDriver.CS[i].MpAxisCyclicSet_0.Error);
//		gDriver.CS[i].Wait[W_CS_COMMANDABORTED]							:= BOOL_TO_DINT(gDriver.CS[i].MpAxisCyclicSet_0.CommandAborted);
//		gDriver.CS[i].Wait[W_CS_COMMANDBUSY]							:= BOOL_TO_DINT(gDriver.CS[i].MpAxisCyclicSet_0.CommandBusy);
//		gDriver.CS[i].Wait[W_CS_UPDATEDONE]								:= BOOL_TO_DINT(gDriver.CS[i].MpAxisCyclicSet_0.UpdateDone);
//		gDriver.CS[i].Wait[W_CS_MOVECYCLICPOSITIONACTIVE]				:= BOOL_TO_DINT(gDriver.CS[i].MpAxisCyclicSet_0.MoveCyclicPositionActive);
//		gDriver.CS[i].Wait[W_CS_MOVECYCLICVELOCITYACTIVE]				:= BOOL_TO_DINT(gDriver.CS[i].MpAxisCyclicSet_0.MoveCyclicVelocityActive);
//		gDriver.CS[i].Wait[W_CS_TORQUECONTROLACTIVE]					:= BOOL_TO_DINT(gDriver.CS[i].MpAxisCyclicSet_0.TorqueControlActive);
//		gDriver.CS[i].Wait[W_CS_TORQUEFEEDFORWARDACTIVE]				:= BOOL_TO_DINT(gDriver.CS[i].MpAxisCyclicSet_0.TorqueFeedForwardActive);
//		gDriver.CS[i].Wait[W_CS_TCAXISLIMITACTIVE]						:= BOOL_TO_DINT(gDriver.CS[i].MpAxisCyclicSet_0.Info.TorqueControl.AxisLimitActive);
//		gDriver.CS[i].Wait[W_CS_TCDATAINITIALIZED]						:= BOOL_TO_DINT(gDriver.CS[i].MpAxisCyclicSet_0.Info.TorqueControl.DataInitialized);
//		gDriver.CS[i].Wait[W_CS_TCINTORQUE]								:= BOOL_TO_DINT(gDriver.CS[i].MpAxisCyclicSet_0.Info.TorqueControl.InTorque);
//		gDriver.CS[i].Wait[W_CS_TCREADY]								:= BOOL_TO_DINT(gDriver.CS[i].MpAxisCyclicSet_0.Info.TorqueControl.Ready);
//		gDriver.CS[i].Wait[W_CS_AXISREADY]								:= BOOL_TO_DINT(gDriver.CS[i].MpAxisCyclicSet_0.Info.AxisReady);
//	END_FOR;

//	gDriver.CS[i].Par.CS.MoveCyclicPosition.Acceleration							//RR
//	gDriver.CS[i].Par.CS.MoveCyclicPosition.AlternativeValueSource					//ENUM
//	gDriver.CS[i].Par.CS.MoveCyclicPosition.Deceleration							//RR
//	gDriver.CS[i].Par.CS.MoveCyclicPosition.DisableJoltLimitation					//ENUM
//	gDriver.CS[i].Par.CS.MoveCyclicPosition.InterpolationMode						//ENUM
//	gDriver.CS[i].Par.CS.MoveCyclicPosition.Jerk									//RR
//	gDriver.CS[i].Par.CS.MoveCyclicPosition.Velocity								//RR
//	gDriver.CS[i].Par.CS.MoveCyclicVelocity.Acceleration							//RR
//	gDriver.CS[i].Par.CS.MoveCyclicVelocity.AlternativeValueSource					//ENUM
//	gDriver.CS[i].Par.CS.MoveCyclicVelocity.Deceleration							//RR
//	gDriver.CS[i].Par.CS.MoveCyclicVelocity.DisableJoltLimitation					//ENUM
//	gDriver.CS[i].Par.CS.MoveCyclicVelocity.InterpolationMode						//ENUM
//	gDriver.CS[i].Par.CS.MoveCyclicVelocity.Jerk									//RR
//	gDriver.CS[i].Par.CS.MoveCyclicVelocity.Mode									//ENUM
//	gDriver.CS[i].Par.CS.TorqueControl.Acceleration									//RR
//	gDriver.CS[i].Par.CS.TorqueControl.CmdIndependentActivation						//BO
//	gDriver.CS[i].Par.CS.TorqueControl.Jerk											//RR
//	gDriver.CS[i].Par.CS.TorqueControl.MaximumVelocity								//RR
//	gDriver.CS[i].Par.CS.TorqueControl.MinimumVelocity								//RR
//	gDriver.CS[i].Par.CS.TorqueControl.Options.CorrectVelocityLimits				//BO
//	gDriver.CS[i].Par.CS.TorqueControl.Options.NoHomingCheck						//BO
//	gDriver.CS[i].Par.CS.TorqueControl.Options.StartAlternativeValueSource			//ENUM
//	gDriver.CS[i].Par.CS.TorqueControl.Options.TimeLimit							//RR
//	gDriver.CS[i].Par.CS.TorqueControl.Options.TorqueAlternativeValueSource			//ENUM
//	gDriver.CS[i].Par.CS.TorqueControl.Options.UseTimeLimit							//BO
//	gDriver.CS[i].Par.CS.TorqueControl.Options.UseVelocityLimits					//BO
//	gDriver.CS[i].Par.CS.TorqueControl.TorqueRamp									//RR
//	gDriver.CS[i].Par.CS.TorqueControl.TorqueResolution								//RR
//	gDriver.CS[i].Par.CS.TorqueFeedForward.InterpolationMode						//ENUM
//	gDriver.CS[i].Par.CS.TorqueFeedForward.Options.DisableMode						//ENUM
//	gDriver.CS[i].Par.CyclicPositionSource											//DINT
//	gDriver.CS[i].Par.CyclicTorqueSource											//DINT
//	gDriver.CS[i].Par.CyclicTorqueFeedForwardSource									//DINT
//	gDriver.CS[i].Par.CyclicVelocitySource											//DINT

END_ACTION
```

#### OMD_OU.st
```iecst
ACTION OMD_OU:

//	FOR i := 0 TO MAX_DRIVER_OU_IDX DO
//		IF NOT gDriver.OU[i].FirstScanComplete THEN
//			gDriver.OU[i].FirstScanComplete 													:= TRUE;
//			gDriver.OU[i].DefaultPar.OU.Acceleration											:= 50.0;							//RR
//
//			brsmemcpy(ADR(gDriver.OU[i].Par),ADR(gDriver.OU[i].DefaultPar),SIZEOF(gDriver.OU[i].Par));
//		END_IF;
//
//		brsmemset(ADR(gDriver.OU[i].Sev),0,SIZEOF(gDriver.OU[i].Sev));
//		brsmemset(ADR(gDriver.OU[i].Status),0,SIZEOF(gDriver.OU[i].Status));
//		FOR j := 0 TO MAX_DRIVER_OU_MON_IDX DO
//			IF gDriver.OU[i].Par.Mon[j].Enable THEN
//				IF gDriver.OU[i].Mon[j] THEN
//					gDriver.OU[i].CTON_Mon[j](IN := TRUE, PT := LREAL_TO_TIME(gDriver.OU[i].Par.Mon[j].Time*1000.0));
//					IF gDriver.OU[i].CTON_Mon[j].Q THEN
//						gDriver.OU[i].Sev[j] := gDriver.OU[i].Par.Mon[j].Sev;
//						IF gDriver.OU[i].Status.Severity < gDriver.OU[i].Sev[j] THEN
//							gDriver.OU[i].Status.Severity := gDriver.OU[i].Sev[j];
//						END_IF;
//					END_IF;
//				ELSE
//					gDriver.OU[i].CTON_Mon[j](IN := FALSE);
//					gDriver.OU[i].Sev[j] := 0;
//				END_IF;
//			ELSE
//				gDriver.OU[i].CTON_Mon[j](IN := FALSE);
//				gDriver.OU[i].Sev[j] := 0;
//			END_IF;
//		END_FOR;
//		IF gDriver.OU[i].Cmd[C_OU_RESET] THEN
//			gDriver.OU[i].Cmd[C_OU_RESET] := FALSE;
//			brsmemset(ADR(gDriver.OU[i].Cmd),0,SIZEOF(gDriver.OU[i].Cmd));
//			brsmemset(ADR(gDriver.OU[i].Sev),0,SIZEOF(gDriver.OU[i].Sev));
//			brsmemset(ADR(gDriver.OU[i].Status),0,SIZEOF(gDriver.OU[i].Status));
//			brsmemcpy(ADR(gDriver.OU[i].Par),ADR(gDriver.OU[i].DefaultPar),SIZEOF(gDriver.OU[i].Par));
//		END_IF;
//		IF gDriver.OU[i].Cmd[C_OU_CLEARCMD] THEN
//			gDriver.OU[i].Cmd[C_OU_CLEARCMD] := FALSE;
//			brsmemset(ADR(gDriver.OU[i].Cmd),0,SIZEOF(gDriver.OU[i].Cmd));
//		END_IF;
//		IF gDriver.OU[i].Cmd[C_OU_CLEARMON] THEN
//			gDriver.OU[i].Cmd[C_OU_CLEARMON] := FALSE;
//			brsmemset(ADR(gDriver.OU[i].Status.Severity),0,SIZEOF(gDriver.OU[i].Status.Severity));
//			brsmemset(ADR(gDriver.OU[i].Sev),0,SIZEOF(gDriver.OU[i].Sev));
//			brsmemset(ADR(gDriver.OU[i].Par.Mon),0,SIZEOF(gDriver.OU[i].Par.Mon));
//		END_IF;
//		IF gDriver.OU[i].Cmd[C_OU_DEFAULTMON] THEN
//			gDriver.OU[i].Cmd[C_OU_DEFAULTMON] := FALSE;
//			brsmemcpy(ADR(gDriver.OU[i].Par.Mon),ADR(gDriver.OU[i].DefaultPar.Mon),SIZEOF(gDriver.OU[i].Par.Mon));
//		END_IF;
//		IF gDriver.OU[i].Cmd[C_OU_CLEARPAR] THEN
//			gDriver.OU[i].Cmd[C_OU_CLEARPAR] := FALSE;
//			brsmemset(ADR(gDriver.OU[i].Par),0,SIZEOF(gDriver.OU[i].Par));
//		END_IF;
//		IF gDriver.OU[i].Cmd[C_OU_DEFAULTPAR] THEN
//			gDriver.OU[i].Cmd[C_OU_DEFAULTPAR] := FALSE;
//			brsmemcpy(ADR(gDriver.OU[i].Par),ADR(gDriver.OU[i].DefaultPar),SIZEOF(gDriver.OU[i].Par));
//		END_IF;
//		gDriver.OU[i].			:= gDriver.OU[i].Cmd[C_OU_ERRORRESET] OR gMain.ErrorReset;
//
//		gDriver.OU[i].Wait[W_OU_NOERROR]				:= BOOL_TO_DOUT(NOT gDriver.OU[i].);
//
//		gDriver.OU[i].Mon[M_OU_ERROR]					:= gDriver.OU[i].MpAxisBasic_0.Error;
//	END_FOR;

//	McSwitchEnum :
//	(
//		mcSWITCH_OFF := 0,		 						(*State/Behavior selection switched off*)
//		mcSWITCH_ON := 1			 					(*State/Behavior selection switched on*)
//	);

END_ACTION
```
